# B&R Automation Studio project 305841_E00002_0 (part 2)

#### PBActions.st
```iecst
// For each button, check the state in the action.
// Call the action regardlesss of sate and check the state
// within the action rather than before calling in case there
// is something to do when the state is off.

// Ready. PB function not assigned
ACTION ProcessPb1 :
  IF owsPendant.PBStates[1] THEN
    // PB state is on ... process away
    ; // nothing to do
  ELSE
    // PB state is off ...
    ; // placeholder for future use
  END_IF;
END_ACTION

// Not assigned
ACTION ProcessPb2 :
  IF owsPendant.PBStates[2] THEN
    // PB state is on ... process away
    ; // nothing to do
  ELSE
    // PB state is off ...
    ; // placeholder for future use
  END_IF;
END_ACTION

// Set Zero
ACTION ProcessPb3 :
  IF owsPendant.PBStates[3] THEN
    // PB state is on ... depending on the axis, home the axis to zero.
    // The PB is a OS, so snapshot the axis selection and the home req.
    // Homing may take several scans, once kicked off, ignore selection
    // changes, PB changes, etc.
    axisSelection := owsPendant.AxisSelection;
    setZeroReq := TRUE;
  ELSE
    // PB state is off ...
    ; // placeholder for future use
  END_IF;
END_ACTION

// Axis Enable
ACTION ProcessPb4 :
  IF owsPendant.PBStates[4] THEN
    // PB state is on ... Send enable if drive is ready to be powered.
    // PB is OneShotted, and request only needs to be set, and is then cleared elsewhere
    axes[owsPendant.AxisSelection].Commands.EnableReq := axes[owsPendant.AxisSelection].Status.IsReadyToPowerOn;
  ELSE
    // PB state is off ...
    ; // placeholder for future use
  END_IF;
END_ACTION

// Axis Disable
ACTION ProcessPb5 :
  IF owsPendant.PBStates[5] THEN
    // PB state is on ... send disable if drive is powered on.
    // PB is OneShotted, and request only needs to be set, and is then cleared elsewhere
    axes[owsPendant.AxisSelection].Commands.DisableReq := axes[owsPendant.AxisSelection].Status.IsPoweredOn;
  ELSE
    // PB state is off ...
    ; // placeholder for future use
  END_IF;
END_ACTION

// Brake Off
ACTION ProcessPb6 :
  IF owsPendant.PBStates[6] THEN
    // PB state is on ... turn on brake release if the drive is disabled
    axes[owsPendant.AxisSelection].Commands.ReleaseBrakeReq := NOT axes[owsPendant.AxisSelection].Status.IsPoweredOn;
  ELSE
    // PB state is off ... turn off brake release
    axes[owsPendant.AxisSelection].Commands.ClearReleaseBrakeReq := TRUE;
    axes[owsPendant.AxisSelection].Commands.ReleaseBrakeReq := FALSE;
  END_IF;
END_ACTION

// Z Set SOC -- Axiz Z needs to be selected
ACTION ProcessPb7 :
  IF owsPendant.PBStates[7] AND owsPendant.AxisSelection = AD_Z THEN
    // PB state is on ... Set the current position to the Start Of Cut (SOC) position as long as the axis is homed.
    IF axes[AD_Z].Status.IsHomed THEN
      gr_CfgCurrent.zAxis.startOfCutPos := axes[AD_Z].Status.Position;
    END_IF;
  ELSE
    // PB state is off ...
    ; // placeholder for future use
  END_IF;
END_ACTION

// Z Set Load/Unload -- Axiz Z needs to be selected
ACTION ProcessPb8 :
  IF owsPendant.PBStates[8] AND owsPendant.AxisSelection = AD_Z THEN
    // PB state is on ... Set the current position to the load/unload position as long as the axis is homed.
    IF axes[AD_Z].Status.IsHomed THEN
      gr_CfgCurrent.zAxis.loadUnloadPos := axes[AD_Z].Status.Position;
    END_IF;
  ELSE
    // PB state is off ...
    ; // placeholder for future use
  END_IF;
END_ACTION

// Not assigned
ACTION ProcessPb9 :
  IF owsPendant.PBStates[9] THEN
    // PB state is on ... process away
    ;
  ELSE
    // PB state is off ...
    ; // placeholder for future use
  END_IF;
END_ACTION

ACTION SetZeroSeq :
  // The set zero sequence is started by PB3.
  // Handle the details here, just to the PB action is kept simple.
  // PB3 sets local axis selection and home req so changes during
  // homing are ignored.

  // Handle the req, and associated OS.
  // The OS is just so we can init values, and not keep resetting them
  // during homing

  IF NOT setZeroReq THEN
    // No Req, clear the OS
    homeSeqOS := FALSE;
  ELSIF setZeroReq AND NOT homeSeqOS THEN
    // Req and no OS, first time thru ...

    // Set the OS
    homeSeqOS := TRUE;

    // Now do the first time setup stuff ...

    // Now set the set zero offset based on the selected axis ... allow for different
    // algorithms based on axis
    IF axisSelection = AD_X THEN
      // TODO: Not sure how to handle X
      axes[axisSelection].MoveParameters.HomeParams.Position := 0.0;
    ELSIF axisSelection = AD_Y THEN
      // TODO: Not sure how to handle Y
      axes[axisSelection].MoveParameters.HomeParams.Position := 0.0;
    ELSIF axisSelection = AD_Z THEN
      // After homing, the desired position is zero + a possible offset
      axes[axisSelection].MoveParameters.HomeParams.Position :=  0.0;
    ELSIF axisSelection = AD_OUTER_ECCENTRIC THEN
      // Outer eccentric just gets homed to 0, no matter where it is, so there is no offset.
      axes[axisSelection].MoveParameters.HomeParams.Position := 0.0;
    ELSIF axisSelection = AD_INNER_ECCENTRIC THEN
      // After homing, the desired position is zero + a possible offset
      axes[axisSelection].MoveParameters.HomeParams.Position :=0.0;
    ELSIF axisSelection = AD_SPINDLE THEN
      // Spindle position isn't critical, so just home to zero
      axes[axisSelection].MoveParameters.HomeParams.Position := 0.0;
    END_IF;

    // Now set the home request for the selected axis
    axes[axisSelection].MoveParameters.HomeParams.Mode := mcHOMING_ABSOLUTE;
    axes[axisSelection].Commands.HomeReq := TRUE;

  ELSIF setZeroReq AND homeSeqOS THEN
    // Req and OS, doing while req is high
    // If the home command and req are both low, the homing is complete, successful or not.
    // If homing is successful, then set the 'isCalibrated' bits.
    IF NOT axes[axisSelection].Commands.HomeReq AND NOT axes[axisSelection].Commands.HomeCmd THEN
      IF axes[axisSelection].Status.IsHomed AND axes[axisSelection].Status.Position = 0.0 THEN
        // Home done and sucessful
        // Set the calibration bits based on selected axis
        IF axisSelection = AD_Z THEN
          gr_PartCurrent.isZCalibrated := TRUE;
        ELSIF axisSelection = AD_OUTER_ECCENTRIC THEN
          gr_PartCurrent.isOutECalibrated := TRUE;
        ELSIF axisSelection = AD_INNER_ECCENTRIC THEN
          gr_PartCurrent.isInECalibrated := TRUE;
        END_IF;
      END_IF;

      // All done, clear the req whether or not it was successful
      setZeroReq := FALSE;
    END_IF;
  END_IF;
END_ACTION

(*
ACTION SetZeroSeqOld :
  // The set zero sequence is started by PB3.
  // Handle the details here, just to the PB action is kept simple.
  // PB3 sets local axis selection and home req so changes during
  // homing are ignored.

  // Handle the req, and associated OS.
  // The OS is just so we can init values, and not keep resetting them
  // during homing

  // The actual homing is handled by the GaMot library function called outside this action.

  IF NOT setZeroReq THEN
    // No Req, clear the OS
    homeSeqOS := FALSE;
  ELSIF setZeroReq AND NOT homeSeqOS THEN
    // Req and no OS, first time thru ...

    // Set the OS
    homeSeqOS := TRUE;

    // Now do the first time setup stuff ...

    // Set the axis to the selected axis
    HomeAxisFb._I_Axis := ADR(axes[axisSelection]);

    // Now set the set zero offset based on the selected axis ... allow for different
    // algorithms based on axis
    IF axisSelection = AD_X THEN
      // TODO: Not sure how to handle X
      HomeAxisFb._I_Position := 0.0;
    ELSIF axisSelection = AD_Y THEN
      // TODO: Not sure how to handle Y
      HomeAxisFb._I_Position := 0.0;
    ELSIF axisSelection = AD_Z THEN
      // After homing, the desired position is zero + a possible offset
      HomeAxisFb._I_Position :=  gr_CfgCurrent.zAxis.setZeroOffset;;
    ELSIF axisSelection = AD_OUTER_ECCENTRIC THEN
      // Outer eccentric just gets homed to 0, no matter where it is, so there is no offset.
      HomeAxisFb._I_Position := 0.0;
    ELSIF axisSelection = AD_INNER_ECCENTRIC THEN
      // After homing, the desired position is zero + a possible offset
      HomeAxisFb._I_Position := gr_CfgCurrent.cuttingHead.setZeroOffset;
    ELSIF axisSelection = AD_SPINDLE THEN
      // Spindle position isn't critical, so just home to zero
      HomeAxisFb._I_Position := 0.0;
    END_IF;

  ELSIF setZeroReq AND homeSeqOS THEN
    // Req and OS, doing while req is high
    // The fb is always called below, and the enable is based on the setZeroReq.
    // Monitor the output of the FB here. It should end sucessfully or in error
    IF fbHomeAbs._O_Done AND NOT fbHomeAbs._O_Error THEN
      // Homing done, and no error -- Success!!
      // Clear the home req and consider the axis homed.
      setZeroReq := FALSE;
      // Set the calibration bits based on selected axis
      IF axisSelection = AD_Z THEN
        gr_PartCurrent.isZCalibrated := TRUE;
      ELSIF axisSelection = AD_OUTER_ECCENTRIC THEN
        gr_PartCurrent.isOutECalibrated := TRUE;
      ELSIF axisSelection = AD_INNER_ECCENTRIC THEN
        gr_PartCurrent.isInECalibrated := TRUE;
      END_IF;
    ELSIF fbHomeAbs._O_Done AND fbHomeAbs._O_Error THEN
      // Homing done, but in error :(
      // Clear the home req
      setZeroReq := FALSE;
      // Clear the calibration bits based on selected axis
      IF axisSelection = AD_Z THEN
        gr_PartCurrent.isZCalibrated := FALSE;
      ELSIF axisSelection = AD_OUTER_ECCENTRIC THEN
        gr_PartCurrent.isOutECalibrated := FALSE;
      ELSIF axisSelection = AD_INNER_ECCENTRIC THEN
        gr_PartCurrent.isInECalibrated := FALSE;
      END_IF;
    ELSE
      // fb not done ... fb must be busy ... nothing to do.
      // Keep for future expansion
      ;
    END_IF;

  END_IF;

END_ACTION

ACTION HomeInPosSeqOld :
  // The home sequence is started by PB3.
  // Handle the details here, just to the PB action is kept simple.
  // PB3 sets local axis selection and home req so changes during
  // homing are ignored.

  // Handle the req, and associated OS.
  // The OS is just so we can init values, and not keep resetting them
  // during homing

  // The actual homing is handled by the GaMot library function called outside this action.

  IF NOT homeInPosReq THEN
    // No Req, clear the OS
    homeSeqOS := FALSE;
  ELSIF homeInPosReq AND NOT homeSeqOS THEN
    // Req and no OS, first time thru ...

    // Set the OS
    homeSeqOS := TRUE;

    // Now do the first time setup stuff ...

    // Set the axis to the selected axis
    fbHomeAbs._I_Axis := ADR(axes[axisSelection]);

    // Now set the desired poition to the axis position
    fbHomeAbs._I_Position := axes[axisSelection].Status.Position;

  ELSIF homeInPosReq AND homeSeqOS THEN
    // Req and OS, doing while req is high
    // The fb is always called below, and the enable is based on the homeInPosReq.
    // Monitor the output of the FB here. It should end sucessfully or in error
    IF fbHomeAbs._O_Done AND NOT fbHomeAbs._O_Error THEN
      // Homing done, and no error -- Success!!
      // Clear the home req and consider the axis homed.
      homeInPosReq := FALSE;

      // Other success stuff here ...

    ELSIF fbHomeAbs._O_Done AND fbHomeAbs._O_Error THEN
      // Homing done, but in error :(
      // Clear the home req
      homeInPosReq := FALSE;

      // Other error stuff here ...

    ELSE
      // fb not done ... fb must be busy ... nothing to do.
      // Keep for future expansion
      ;
    END_IF;

  END_IF;

 END_ACTION
*)
```

### Program Logical/PlcLogic/CuttingFluidVFD (IEC)

#### Variables.var
```iecst
VAR

  almMask : UDINT;
  tmrCfFlowOk : TON; (* flow established timer *)
  timeCfFlowOk : TIME;

END_VAR
```

#### Action.st
```iecst
ACTION ProcessAlarms :
  // Alarm Enable/disable. These are permanent, but include here to easily make them dynamic.
  // Tank level
  gr_AI_LT_CFTankLevel_Params.AlmEnable := FALSE; // not fitted.
  // Flow
  gr_AI_FT_CFFlow_Params.AlmEnable := FALSE; // not fitted
  // Level switch
  gr_DI_LSL_CFTank_Params.AlmEnable := FALSE; // not fitted
  // Locator
  gr_DI_ZS_CFTankLocator_Params.AlmEnable:= TRUE;

  // Pressure and flow sensors -- enable while pump is running
  gr_AI_PT_CFPumpOutlet_Params.AlmEnable := cfVfd.isRunning;
  gr_AI_PT_CFFilterOutlet_Params.AlmEnable := cfVfd.isRunning;
  gr_AI_DP_CFFilter_Params.AlmEnable := cfVfd.isRunning;
  gr_AI_FT_CFFlow_Params.AlmEnable := cfVfd.isRunning;

  // Put alarm status into structure
  // isLocated
  cfVfd.isLocated := DI_ZS_CFTankLocator.alms = GAPIO_ALARM_NONE;

  // Level switch
  cfVfd.isAlmLoLvlSw := DI_LSL_CFTank.alms <> GAPIO_ALARM_NONE;

  // Flow
  // consider alarm on range, channel or lo lo alms
  almMask := 	GAPIO_ALARM_RANGEHI OR GAPIO_ALARM_RANGELO OR GAPIO_ALARM_CHANNEL OR GAPIO_ALARM_LOLO;
  cfVfd.isAlmLoFlow := (AI_FT_CFFlow.alms AND almMask) <> 0;
  // consider warning on lo alm
  almMask := GAPIO_ALARM_LO;
  cfVfd.isWarnLoFlow := (AI_FT_CFFlow.alms AND almMask) <> 0;

  // Fluid Level
  // consider alarm on range, channel or lo lo alms
  almMask := 	GAPIO_ALARM_RANGEHI OR GAPIO_ALARM_RANGELO OR GAPIO_ALARM_CHANNEL OR GAPIO_ALARM_LOLO;
  cfVfd.isAlmLoFluid := (AI_LT_CFTankLevel.alms AND almMask) <> 0;
  // consider warning on lo alm
  almMask := 	GAPIO_ALARM_LO;
  cfVfd.isWarnLoFluid := (AI_LT_CFTankLevel.alms AND almMask) <> 0;

  // Pump Outlet pressure
  // consider alarm on hi range, channel or hi hi alms
  almMask := 	GAPIO_ALARM_RANGEHI OR GAPIO_ALARM_CHANNEL OR GAPIO_ALARM_HIHI;
  cfVfd.isAlmHiOutletPressure := (AI_PT_CFPumpOutlet.alms AND almMask) <> 0;
  // consider alarm on range, channel or lo lo alms
  almMask := 	GAPIO_ALARM_RANGELO OR GAPIO_ALARM_LOLO;
  cfVfd.isAlmLoOutletPressure := (AI_PT_CFPumpOutlet.alms AND almMask) <> 0;
  // consider warning on lo alm
  almMask := 	GAPIO_ALARM_LO;
  cfVfd.isWarnLoOutletPressure := (AI_PT_CFPumpOutlet.alms AND almMask) <> 0;
  // consider warning on hi alm
  almMask := 	GAPIO_ALARM_HI;
  cfVfd.isWarnHiOutletPressure := (AI_PT_CFPumpOutlet.alms AND almMask) <> 0;

  // Hi Filter DP -- channel and range will trigger hi and low
  almMask := 	GAPIO_ALARM_RANGEHI OR GAPIO_ALARM_RANGELO OR GAPIO_ALARM_CHANNEL OR GAPIO_ALARM_HI;
  cfVfd.isWarnHiFilterDp := (AI_DP_CFFilter.alms AND almMask) <> 0;
  // Lo Filter DP -- channel and range will trigger hi and low
  almMask := 	GAPIO_ALARM_RANGEHI OR GAPIO_ALARM_RANGELO OR GAPIO_ALARM_CHANNEL OR GAPIO_ALARM_LO;
  cfVfd.isWarnLoFilterDp := (AI_DP_CFFilter.alms AND almMask) <> 0;

  // Alarm and warning summaries
  cfVfd.isWarnSummary := cfVfd.isWarnLoFlow OR cfVfd.isWarnLoFluid OR
  cfVfd.isWarnLoOutletPressure OR cfVfd.isWarnHiOutletPressure OR
  cfVfd.isWarnLoFilterDp OR cfVfd.isWarnHiFilterDp;

  cfVfd.isAlmSummary := cfVfd.isAlmLoFlow OR cfVfd.isAlmLoLvlSw OR
  cfVfd.isAlmLoFluid OR cfVfd.isAlmLoOutletPressure OR cfVfd.isAlmHiOutletPressure;

END_ACTION
```

#### Main.st
```iecst
PROGRAM _INIT

  // Flow established time
  timeCfFlowOk := T#5s;

END_PROGRAM

PROGRAM _CYCLIC

  // Process the alarms
  ProcessAlarms;

  cfVfd.isAllowedToStart :=
    (operatingMode.OperatingMode = OM_MANUAL_MODE OR
    operatingMode.OperatingMode = OM_PENDANT_MODE OR
    operatingMode.OperatingMode = OM_PRODUCTION_MODE) AND
    axes[AD_CF_VFD].Status.IsPoweredOn AND
    axes[AD_CF_VFD].Status.IsHomed AND
    cfVfd.isLocated AND
    NOT cfVfd.isAlmLoLvlSw AND NOT cfVfd.isAlmLoFluid;

  cfVfd.isAllowedToRun :=
    (operatingMode.OperatingMode = OM_MANUAL_MODE OR
    operatingMode.OperatingMode = OM_PENDANT_MODE OR
    operatingMode.OperatingMode = OM_PRODUCTION_MODE) AND
    axes[AD_CF_VFD].Status.IsPoweredOn AND
    axes[AD_CF_VFD].Status.IsHomed AND
    cfVfd.isLocated AND
    NOT cfVfd.isAlmLoLvlSw AND NOT cfVfd.isAlmLoFluid AND
    NOT cfVfd.isAlmLoFlow AND NOT cfVfd.isAlmLoOutletPressure AND
    NOT cfVfd.isAlmHiOutletPressure;

  // Map the axis status to the cf structure to get a running bit
  cfVfd.isRunning := axes[AD_CF_VFD].Status.IsMoveActive;

  // Determine when good flow is established -- time delay no flow problems
  tmrCfFlowOk(IN:= cfVfd.isRunning AND NOT cfVfd.isAlmLoFlow, PT:= timeCfFlowOk);
  cfVfd.isFlowEstablished := tmrCfFlowOk.Q;

END_PROGRAM

PROGRAM _EXIT
	(* Insert code here *)

END_PROGRAM
```

### Program Logical/PlcLogic/OmSafeDev (IEC) - Operating Mode State Machine

#### OmSafeDev.typ - Local data types
```iecst
TYPE
  (* Machine specific HMI axis requests. Intended to have one of these structures per axis. *)
  sHmiAxisReqs : STRUCT
    (* Boolean requests in this section. *)
    (* (none *)
    (* numerical requests *)
    (* (none *)
    (* hmi move type and direction selection related *)
    absMoveEnable : BOOL := TRUE; (* allow move type selection by default *)
    relMoveEnable : BOOL := TRUE;
    velMoveEnable : BOOL := TRUE;
    directionPosEnable : BOOL := TRUE; (* allow direction selection by default *)
    directionNegEnable : BOOL := TRUE;
    directionShortestEnable : BOOL := TRUE;
    moveDistanceEnable : BOOL := TRUE; (* enable params by default *)
    movePositionEnable : BOOL := TRUE;
    shiftEnable : BOOL := FALSE; (* coordinated axis shift enabled *)
    moveDesignation: DINT := -1; (* -1 is no selection *)
    direction: DINT := -1; (* -1 is no selection *)
    (* axis designation. Two different data types for convenience. *)
    axisNo : USINT := 0; (* default to initial so setting a value can be detected. USINT for easy use in loops *)
    axisDesignation : eAXIS_DESIGNATION := AD_UNKNOWN; (* default to initial so setting a value can be detected *)
  END_STRUCT;

  (* Machine specific HMI process requests. Intended to have one of these per machine or otherwise as needed, but not per axis. *)
  sHmiProcessReqs : STRUCT
    (* Boolean requests in this section. *)
    (* NOTE/CAUTION These request bits may get cleared/copied by memcpy/memclr
    So be careful about adding boolean requests outside of this section.
    See ClearManualReqs action for example, in OmSaveDev program.
    Bool requests above zReqMoveUpLimit won't get auto cleared *)
    zReqMoveUpLimit : BOOL := FALSE;
    zReqMoveDownLimit : BOOL := FALSE;
    zReqMoveLoadUnload : BOOL := FALSE;
    zReqMoveSoc : BOOL := FALSE;
    cuttingHeadMoveReqRetract : BOOL := FALSE;
    (* NOTE/CAUTION Bool requests below cuttingHeadMoveReqRetract won't get auto cleared *)
    (* numerical requests *)
    cuttingHeadReqDepth : LREAL := 0.0;
  END_STRUCT;

END_TYPE
```

#### OmSafeDev.var - Local variables
```iecst
VAR CONSTANT

END_VAR

VAR

  (* info from safety controller *)
  fs_AllSMsOk : BOOL;
  fs_EmoCmd : BOOL; (* H:Ok, L:EMO *)
  fs_EmoOwsActive : BOOL; (* H:Ok, L: EMO *)
  fs_EmoOwsOk : BOOL; (* H:Wiring Ok, L:Error *)
  fs_InSafeMode : BOOL; (* H:InSafeMode, L: Not in safe mode *)
  fs_KeyswitchInRun : BOOL; (* H:Run Pos, L: Not in run pos *)
  fs_KeyswitchOk : BOOL; (* H:Wiring Ok, L:Error *)
  fs_StartPbActive : BOOL; (* H:Start Req, L: Not pressed *)
  fs_StartPbOk : BOOL; (* H:Wiring Ok, L:Error *)
  fs_StopPbActive : BOOL; (* H: Allow Run, L: Stop *)
  fs_StopPbOk : BOOL; (* H:Wiring Ok, L:Error *)
  fs_CfGateClosed : BOOL; (* H:Closed, L: Open *)
  fs_CfGateClosedLocked : BOOL; (* H:Closed and locked(Ok), L: Open and/or unlocked *)
  fs_CfGateClosedOk : BOOL; (* H:Wiring Ok, L: Error *)

  (* info to safety controller *)
  ts_ResetEStop : BOOL;
  ts_ResetSafeMC : BOOL;
  ts_InEmoMode : BOOL;
  ts_InSafeMode : BOOL;
  ts_InPendantMode : BOOL;

  (* cycle start/stop req *)
  tmrReqStartPulse : TP;
  tmrReqStopPulse : TP;

  (* EMO Reset *)
  timeEStopResetAllow : TIME;
  eStopResetAllowSecRemain : DINT;
  tmrEStopResetAllow : TON;
  timeResetPulse : TIME;
  tmrResetPulse : TP;

  (* HMI process specific, machine specific, and axis requests *)
  hmiProcessReqs : sHmiProcessReqs; (* process specific reqs *)
  hmiMachineAxisReqs : ARRAY[0..AXIS_COUNT] OF sHmiAxisReqs; (* machine specific requests that get turned into library reqs *)
  hmiLibraryAxisReqs : ARRAY[0..AXIS_COUNT] OF sMot_HmiAxisReqs; (* standard/basic requests handled by the library *)

  (* pointers used for memcpy/memset *)
  pSrc :  UDINT;
  pDest :  UDINT;
  byteCount :  UDINT;
  nxtAddr :  UDINT;

  (* axis index *)
  axisNo : DINT;

  (* fb to process Reqs *)
  procHmiProcessReqs : fbHandleHmiProcessReqs;
  procManualAxisReqsSpindle : fbHandleHmiAxisReq;
  procManualAxisReqsOutE : fbHandleHmiAxisReq;
  procManualAxisReqsInE : fbHandleHmiAxisReq;
  procManualAxisReqsZ : fbHandleHmiAxisReq;
  procManualAxisReqsHw : fbHandleHmiAxisReq;
  procManualAxisReqsCfVfd : fbHandleHmiAxisReq;
END_VAR
```

#### Init.st
```iecst
PROGRAM _INIT

  // TODO: Security levels. For now just set as operator so OM SM can be programmed
  operatingMode.SecurityLevel := SL_OPERATOR;

  // EMO Reset time
  timeEStopResetAllow := T#10s;
  timeResetPulse := T#1s;

  // Init to create variables
  // If values are only mapped, and not used in logic anywhere, the compiler does not
  // create them. They are not available to
  // the HMI, and the compiler also complains about
  // them being declared but not used
  fs_AllSMsOk := FALSE;
  fs_EmoCmd := FALSE;
  fs_EmoOwsActive := FALSE;
  fs_EmoOwsOk := FALSE;
  // pendant signals are mapped into pendant structure
  // fs_EmoPendantActive := FALSE;
  // fs_EmoPendantOk := FALSE;
  // fs_AllowPendantMoves := FALSE;
  fs_KeyswitchInRun := FALSE;
  fs_KeyswitchOk := FALSE;
  fs_InSafeMode := FALSE;
  fs_StartPbActive := FALSE;
  fs_StartPbOk := FALSE;
  fs_StopPbActive := FALSE;
  fs_StopPbOk := FALSE;
  fs_CfGateClosedLocked := FALSE;
  fs_CfGateClosedOk := FALSE;

  ts_ResetEStop := FALSE;
  ts_ResetSafeMC := FALSE;

  // Init process req fb
  procHmiProcessReqs._I_ProcessReqs := ADR(hmiProcessReqs);
  procHmiProcessReqs._I_pLibraryAxesReqs:= ADR(hmiLibraryAxisReqs); // Start of array of sMot_HmiAxisReqs

  // Init manual mode requests
  hmiLibraryAxisReqs[AD_SPINDLE].axisNo := DINT_TO_USINT(AD_SPINDLE);
  hmiMachineAxisReqs[AD_SPINDLE].axisNo := DINT_TO_USINT(AD_SPINDLE);
  hmiMachineAxisReqs[AD_SPINDLE].axisDesignation := AD_SPINDLE;
  procManualAxisReqsSpindle._I_Axis := ADR(axes[AD_SPINDLE]);
  procManualAxisReqsSpindle._I_SlaveAxis := ADR(axes[axes[AD_SPINDLE].CouplingParameters.SlaveAxisNo]);
  procManualAxisReqsSpindle._I_LibraryAxisReqs := ADR(hmiLibraryAxisReqs[AD_SPINDLE]);
  procManualAxisReqsSpindle._I_MachineAxisReqs := ADR(hmiMachineAxisReqs[AD_SPINDLE]);
  procManualAxisReqsSpindle._I_AxisPositionLimits := ADR(gr_AxisPositionLimits[AD_SPINDLE]);

  // Outer Eccentric
  hmiLibraryAxisReqs[AD_OUTER_ECCENTRIC].axisNo := DINT_TO_USINT(AD_OUTER_ECCENTRIC);
  hmiMachineAxisReqs[AD_OUTER_ECCENTRIC].axisNo := DINT_TO_USINT(AD_OUTER_ECCENTRIC);
  hmiMachineAxisReqs[AD_OUTER_ECCENTRIC].axisDesignation := AD_OUTER_ECCENTRIC;
  procManualAxisReqsOutE._I_Axis := ADR(axes[AD_OUTER_ECCENTRIC]);
  procManualAxisReqsOutE._I_SlaveAxis := ADR(axes[axes[AD_OUTER_ECCENTRIC].CouplingParameters.SlaveAxisNo]);
  procManualAxisReqsOutE._I_LibraryAxisReqs := ADR(hmiLibraryAxisReqs[AD_OUTER_ECCENTRIC]);
  procManualAxisReqsOutE._I_MachineAxisReqs:= ADR(hmiMachineAxisReqs[AD_OUTER_ECCENTRIC]);
  procManualAxisReqsOutE._I_AxisPositionLimits := ADR(gr_AxisPositionLimits[AD_OUTER_ECCENTRIC]);

  // Inner Eccentric
  hmiLibraryAxisReqs[AD_INNER_ECCENTRIC].axisNo := DINT_TO_USINT(AD_INNER_ECCENTRIC);
  hmiMachineAxisReqs[AD_INNER_ECCENTRIC].axisNo := DINT_TO_USINT(AD_INNER_ECCENTRIC);
  hmiMachineAxisReqs[AD_INNER_ECCENTRIC].axisDesignation := AD_INNER_ECCENTRIC;
  procManualAxisReqsInE._I_Axis := ADR(axes[AD_INNER_ECCENTRIC]);
  procManualAxisReqsInE._I_SlaveAxis := ADR(axes[axes[AD_INNER_ECCENTRIC].CouplingParameters.SlaveAxisNo]);
  procManualAxisReqsInE._I_LibraryAxisReqs := ADR(hmiLibraryAxisReqs[AD_INNER_ECCENTRIC]);
  procManualAxisReqsInE._I_MachineAxisReqs := ADR(hmiMachineAxisReqs[AD_INNER_ECCENTRIC]);
  procManualAxisReqsInE._I_AxisPositionLimits := ADR(gr_AxisPositionLimits[AD_INNER_ECCENTRIC]);

  // Z
  hmiLibraryAxisReqs[AD_Z].axisNo := DINT_TO_USINT(AD_Z);
  hmiMachineAxisReqs[AD_Z].axisNo := DINT_TO_USINT(AD_Z);
  hmiMachineAxisReqs[AD_Z].axisDesignation := AD_Z;
  procManualAxisReqsZ._I_Axis := ADR(axes[AD_Z]);
  procManualAxisReqsZ._I_SlaveAxis := ADR(axes[axes[AD_Z].CouplingParameters.SlaveAxisNo]);
  procManualAxisReqsZ._I_LibraryAxisReqs := ADR(hmiLibraryAxisReqs[AD_Z]);
  procManualAxisReqsZ._I_MachineAxisReqs := ADR(hmiMachineAxisReqs[AD_Z]);
  procManualAxisReqsZ._I_AxisPositionLimits := ADR(gr_AxisPositionLimits[AD_Z]);

  // Handwheel (Axis 7)
  hmiLibraryAxisReqs[AD_HANDWHEEL].axisNo := DINT_TO_USINT(AD_HANDWHEEL);
  hmiMachineAxisReqs[AD_HANDWHEEL].axisNo := DINT_TO_USINT(AD_HANDWHEEL);
  hmiMachineAxisReqs[AD_HANDWHEEL].axisDesignation := AD_HANDWHEEL;
  procManualAxisReqsHw._I_Axis := ADR(axes[AD_HANDWHEEL]);
  procManualAxisReqsHw._I_SlaveAxis := ADR(axes[axes[AD_HANDWHEEL].CouplingParameters.SlaveAxisNo]);
  procManualAxisReqsHw._I_LibraryAxisReqs := ADR(hmiLibraryAxisReqs[AD_HANDWHEEL]);
  procManualAxisReqsHw._I_MachineAxisReqs := ADR(hmiMachineAxisReqs[AD_HANDWHEEL]);
  procManualAxisReqsHw._I_AxisPositionLimits := ADR(gr_AxisPositionLimits[AD_HANDWHEEL]);

  // Cutting fluid VFD (Axis 8)
  hmiLibraryAxisReqs[AD_CF_VFD].axisNo := DINT_TO_USINT(AD_CF_VFD);
  hmiMachineAxisReqs[AD_CF_VFD].axisNo := DINT_TO_USINT(AD_CF_VFD);
  hmiMachineAxisReqs[AD_CF_VFD].axisDesignation := AD_CF_VFD;
  procManualAxisReqsCfVfd._I_Axis := ADR(axes[AD_CF_VFD]);
  procManualAxisReqsCfVfd._I_SlaveAxis := ADR(axes[axes[AD_CF_VFD].CouplingParameters.SlaveAxisNo]);
  procManualAxisReqsCfVfd._I_LibraryAxisReqs := ADR(hmiLibraryAxisReqs[AD_CF_VFD]);
  procManualAxisReqsCfVfd._I_MachineAxisReqs := ADR(hmiMachineAxisReqs[AD_CF_VFD]);
  procManualAxisReqsCfVfd._I_AxisPositionLimits := ADR(gr_AxisPositionLimits[AD_CF_VFD]);

  // Clear reqs that may result in motion or physical changes to an axis
  ClearMotionReqs;
  // Clear other requests
  ClearNonMotionReqs;

END_PROGRAM
```

#### OmSafeDev.sfc - Cyclic code
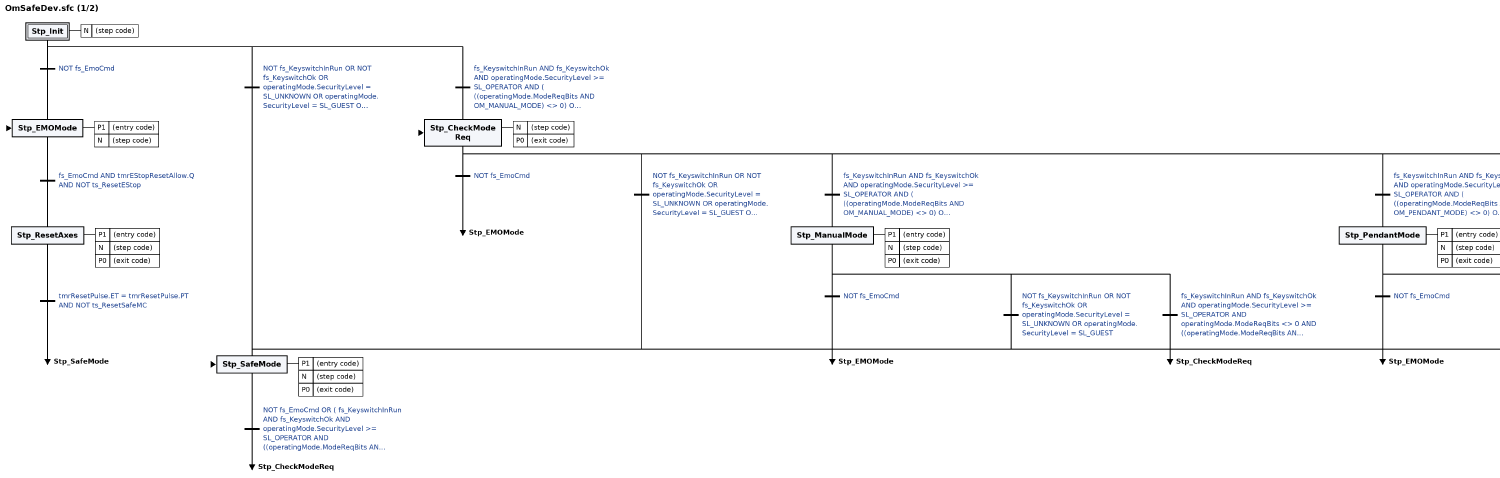
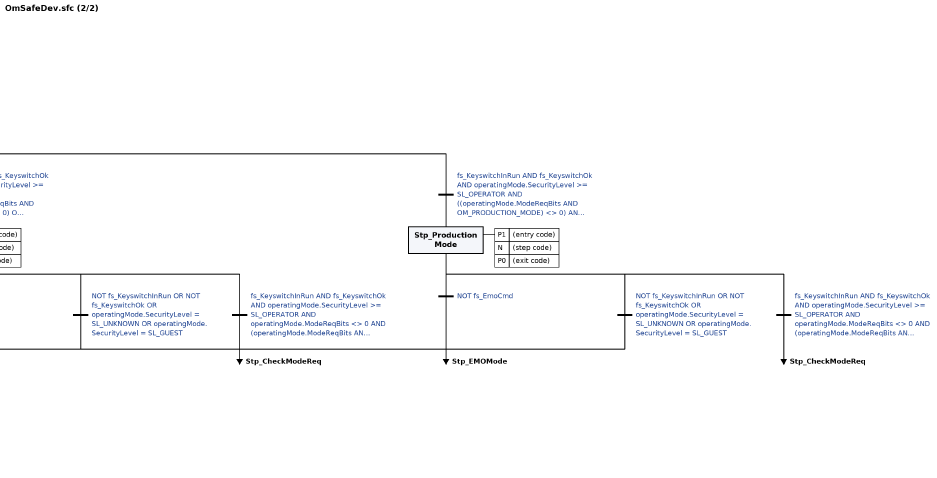
```iecst
PROGRAM _CYCLIC
INITIAL_STEP Stp_Init:
// Set Operating State
operatingMode.OperatingMode := OM_INITIAL;

END_STEP
TRANSITION EMO Cmd FROM Stp_Init TO Stp_EMOMode:=
// EStop command from safety plc H:Ok, L:EMO
NOT fs_EmoCmd
END_TRANSITION
TRANSITION keyswich in safe, not ok or bad SL or no mode req FROM Stp_Init TO Stp_SafeMode:=
// Keyswitch not in run or not okay
NOT fs_KeyswitchInRun OR
NOT fs_KeyswitchOk OR
// or not adequate security level
operatingMode.SecurityLevel = SL_UNKNOWN OR
operatingMode.SecurityLevel = SL_GUEST OR
// Or a mode isnt' being requested.
// Go to safe initially if all else is okay so a mode must be chosen
operatingMode.ModeReqBits = 0
END_TRANSITION
TRANSITION keyswitch in run and SL FROM Stp_Init TO Stp_CheckModeReq:=
// Keyswitch in run and adequate security level
fs_KeyswitchInRun AND
fs_KeyswitchOk AND
operatingMode.SecurityLevel >= SL_OPERATOR AND
// and a mode is requested
(
((operatingMode.ModeReqBits AND OM_MANUAL_MODE) <> 0) OR
((operatingMode.ModeReqBits AND OM_PENDANT_MODE) <> 0) OR
((operatingMode.ModeReqBits AND OM_PRODUCTION_MODE) <> 0)
)

END_TRANSITION
STEP Stp_CheckModeReq:
// This is a transition state. The state machine should not stay here, so don't
// set the mode upon entry. The mode in fact cannot be changed, as the current value is
// is used to transition back into the same state if a request was made but not granted
// for example production mode req but gate isn't shut.

// Clear reqs that may result in motion or physical changes to an axis
ClearMotionReqs;
// Clear other requests
ClearNonMotionReqs;

// Axis permit and other permissives
OtherModeAxisPermits;
ModeIndependentPermissions;
END_STEP
EXIT_ACTION
// Clear the request bits when leaving
operatingMode.ModeReqBits := 0;
END_ACTION
TRANSITION EMO Cmd FROM Stp_CheckModeReq TO Stp_EMOMode:=
// EStop command from safety plc H:Ok, L:EMO
NOT fs_EmoCmd
END_TRANSITION
(* @SFCISJUMP := 'Stp_EMOMode' *)
TRANSITION key not in run or bad SL or prod mode but not allowed FROM Stp_CheckModeReq TO Stp_SafeMode:=
// Keyswitch not in run or not okay, or not adequate security level
NOT fs_KeyswitchInRun OR
NOT fs_KeyswitchOk OR
operatingMode.SecurityLevel = SL_UNKNOWN OR
operatingMode.SecurityLevel = SL_GUEST OR
// or requested production mode but the gate isn't closed, so stay here in safe mode
(((operatingMode.ModeReqBits AND OM_PRODUCTION_MODE) <> 0) AND NOT fs_CfGateClosed AND operatingMode.OperatingMode = OM_SAFE_MODE)

END_TRANSITION
TRANSITION req manual mode or prod mode but not allowed FROM Stp_CheckModeReq TO Stp_ManualMode:=
// Keyswitch in run and adequate security level
fs_KeyswitchInRun AND
fs_KeyswitchOk AND
operatingMode.SecurityLevel >= SL_OPERATOR AND
(
// Req Manual Mode
((operatingMode.ModeReqBits AND OM_MANUAL_MODE) <> 0) OR
// or requested production mode but the gate isn't closed, so stay here in manual mode
(((operatingMode.ModeReqBits AND OM_PRODUCTION_MODE) <> 0) AND NOT fs_CfGateClosed AND operatingMode.OperatingMode = OM_MANUAL_MODE)
)

END_TRANSITION
STEP Stp_ManualMode:
// Block mode request for current mode, but keep the others
// This prevents it from being seen as a request
operatingMode.ModeReqBits := operatingMode.ModeReqBits AND NOT OM_MANUAL_MODE; (* bit 4 clear *)

// Axis permit and other permissives
ManualModeAxisPermits;
ModeIndependentPermissions;

// Pulse the Reset SafeMC on request.
// This allows the reset of the safety enable instructions in the
// SafePLC while the system is not in EMO mode.
// The SafeMC reset sometimes isn't effective unless the axis is otherwise allowed to be powered.
tmrResetPulse(IN:= operatingMode.ReqEmoReset);
ts_ResetSafeMC := tmrResetPulse.Q;
operatingMode.ReqEmoReset := FALSE;

// Clear production start/stop cycle
operatingMode.ReqCycleStart := FALSE;
operatingMode.ReqCycleStop := FALSE;
operatingMode.HmiReqCycleStart := FALSE;
operatingMode.HmiReqCycleStop:= FALSE;

// Process manual requests
// Inputs set in init. This fb looks for a rising edge on the HMI move request, and
// one-shots the axis move requests. It is inteneded to be run on every scan,
// at least while in manual mode.
procManualAxisReqsSpindle();
procManualAxisReqsOutE();
procManualAxisReqsInE();
procManualAxisReqsZ();
procManualAxisReqsHw();
procManualAxisReqsCfVfd();
END_STEP
ENTRY_ACTION
// Set Operating State
operatingMode.OperatingMode := OM_MANUAL_MODE;
// To Safety PLC
ts_InManualMode := TRUE;

// Reset pulse timer
tmrResetPulse(IN:= FALSE, PT:= timeResetPulse);

// Clear reqs that may result in motion or physical changes to an axis
ClearMotionReqs;
// Clear other requests
ClearNonMotionReqs;

// Init fb with low reqs so rising edge detection is ready
procManualAxisReqsSpindle();
procManualAxisReqsOutE();
procManualAxisReqsInE();
procManualAxisReqsZ();
procManualAxisReqsHw();
procManualAxisReqsCfVfd();
END_ACTION
EXIT_ACTION
// To Safety PLC
ts_InManualMode := FALSE;

// Clear reqs that may result in motion or physical changes to an axis
ClearMotionReqs;
// Clear other requests
ClearNonMotionReqs;

// Init fb with low reqs so rising edge detection is ready
procManualAxisReqsSpindle();
procManualAxisReqsOutE();
procManualAxisReqsInE();
procManualAxisReqsZ();
procManualAxisReqsHw();
procManualAxisReqsCfVfd();
END_ACTION
TRANSITION EMO Cmd FROM Stp_ManualMode TO Stp_EMOMode:=
// EStop command from safety plc H:Ok, L:EMO
NOT fs_EmoCmd
END_TRANSITION
(* @SFCISJUMP := 'Stp_EMOMode' *)
TRANSITION key not in run or bad SL FROM Stp_ManualMode TO Stp_SafeMode:=
// Keyswitch not in run or not okay, or not adequate security level
NOT fs_KeyswitchInRun OR
NOT fs_KeyswitchOk OR
operatingMode.SecurityLevel = SL_UNKNOWN OR
operatingMode.SecurityLevel = SL_GUEST
END_TRANSITION
TRANSITION req mode change FROM Stp_ManualMode TO Stp_CheckModeReq:=
// Keyswitch in run and adequate security level
fs_KeyswitchInRun AND
fs_KeyswitchOk AND
operatingMode.SecurityLevel >= SL_OPERATOR AND
// Req mode change (req other than current mode)
operatingMode.ModeReqBits <> 0 AND
((operatingMode.ModeReqBits AND OM_MANUAL_MODE) = 0)

END_TRANSITION
(* @SFCISJUMP := 'Stp_CheckModeReq' *)
TRANSITION req pendant mode or prod mode but not allowed FROM Stp_CheckModeReq TO Stp_PendantMode:=
// Keyswitch in run and adequate security level
fs_KeyswitchInRun AND
fs_KeyswitchOk AND
operatingMode.SecurityLevel >= SL_OPERATOR AND
(
// Req Pendant Mode
((operatingMode.ModeReqBits AND OM_PENDANT_MODE) <> 0) OR
// or requested production mode but the gate isn't closed, so stay here in pendant mode
(((operatingMode.ModeReqBits AND OM_PRODUCTION_MODE) <> 0) AND NOT fs_CfGateClosed AND operatingMode.OperatingMode = OM_PENDANT_MODE)
)

END_TRANSITION
STEP Stp_PendantMode:
// Block mode request for current mode, but keep the others
// This prevents it from being seen as a request
operatingMode.ModeReqBits := operatingMode.ModeReqBits AND NOT OM_PENDANT_MODE; (* bit 5 clear *)

// Axis permit and other permissives
PendantModeAxisPermits;
ModeIndependentPermissions;

// Clear process reqs
ClearProcessReqs;

// Pulse the Reset SafeMC on request.
// This allows the reset of the safety enable instructions in the
// SafePLC while the system is not in EMO mode.
// The SafeMC reset sometimes isn't effective unless the axis is otherwise allowed to be powered.
tmrResetPulse(IN:= operatingMode.ReqEmoReset);
ts_ResetSafeMC := tmrResetPulse.Q;
operatingMode.ReqEmoReset := FALSE;

// Clear production start/stop cycle
operatingMode.ReqCycleStart := FALSE;
operatingMode.ReqCycleStop := FALSE;
operatingMode.HmiReqCycleStart := FALSE;
operatingMode.HmiReqCycleStop:= FALSE;

// Use the gear ratio coming from the pendant for the hmi request strucure.
// It is the hmi request structure values that will get sent to the axis.
hmiLibraryAxisReqs[AD_HANDWHEEL].gearRatioNumerator := owsPendant.GearRatioNumerator;
hmiLibraryAxisReqs[AD_HANDWHEEL].gearRatioDenominator := owsPendant.GearRatioDenominator;

// Process manual requests -- Allow these in pendant mode.
// Inputs set in init. This fb looks for a rising edge on the HMI move request, and
// one-shots the axis move requests. It is inteneded to be run on every scan,
// at least while in manual mode.
procManualAxisReqsSpindle();
procManualAxisReqsOutE();
procManualAxisReqsInE();
procManualAxisReqsZ();
procManualAxisReqsHw();
procManualAxisReqsCfVfd();

END_STEP
ENTRY_ACTION
// Set Operating State
operatingMode.OperatingMode := OM_PENDANT_MODE;
// To Safety PLC
ts_InPendantMode := TRUE;

// Reset pulse timer
tmrResetPulse(IN:= FALSE, PT:= timeResetPulse);

// Disable enabled axes on entry into pendant mode -- allows starting from the same point
FOR axisNo := 1 TO AXIS_COUNT DO
  axes[axisNo].Commands.DisableReq := axes[axisNo].Status.IsPoweredOn;
END_FOR;

// Clear reqs that may result in motion or physical changes to an axis
ClearMotionReqs;
// Clear other requests
ClearNonMotionReqs;

// Init fb with low reqs so rising edge detection is ready
procManualAxisReqsSpindle();
procManualAxisReqsOutE();
procManualAxisReqsInE();
procManualAxisReqsZ();
procManualAxisReqsHw();
procManualAxisReqsCfVfd();

END_ACTION
EXIT_ACTION
// To Safety PLC
ts_InPendantMode := FALSE;

// Clear reqs that may result in motion or physical changes to an axis
ClearMotionReqs;
// Clear other requests
ClearNonMotionReqs;

// Init fb with low reqs so rising edge detection is ready
procManualAxisReqsSpindle();
procManualAxisReqsOutE();
procManualAxisReqsInE();
procManualAxisReqsZ();
procManualAxisReqsHw();
procManualAxisReqsCfVfd();
END_ACTION
TRANSITION EMO Cmd FROM Stp_PendantMode TO Stp_EMOMode:=
// EStop command from safety plc H:Ok, L:EMO
NOT fs_EmoCmd
END_TRANSITION
(* @SFCISJUMP := 'Stp_EMOMode' *)
TRANSITION key not in run or bad SL FROM Stp_PendantMode TO Stp_SafeMode:=
// Keyswitch not in run or not okay, or not adequate security level
NOT fs_KeyswitchInRun OR
NOT fs_KeyswitchOk OR
operatingMode.SecurityLevel = SL_UNKNOWN OR
operatingMode.SecurityLevel = SL_GUEST
END_TRANSITION
TRANSITION req mode change FROM Stp_PendantMode TO Stp_CheckModeReq:=
// Keyswitch in run and adequate security level
fs_KeyswitchInRun AND
fs_KeyswitchOk AND
operatingMode.SecurityLevel >= SL_OPERATOR AND
// Req mode change (req other than current mode)
operatingMode.ModeReqBits <> 0 AND
(operatingMode.ModeReqBits AND OM_PENDANT_MODE) = 0

END_TRANSITION
(* @SFCISJUMP := 'Stp_CheckModeReq' *)
TRANSITION req production mode FROM Stp_CheckModeReq TO Stp_ProductionMode:=
// Keyswitch in run and adequate security level
fs_KeyswitchInRun AND
fs_KeyswitchOk AND
operatingMode.SecurityLevel >= SL_OPERATOR AND
// Req Production Mode
((operatingMode.ModeReqBits AND OM_PRODUCTION_MODE) <> 0) AND
// gate must be closed for production mode
fs_CfGateClosed
END_TRANSITION
STEP Stp_ProductionMode:
// Block mode request for current mode, but keep the others
// This prevents it from being seen as a request
operatingMode.ModeReqBits := operatingMode.ModeReqBits AND NOT OM_PRODUCTION_MODE; (* bit 6 clear *)

// Axis permit and other permissives
ProductionModeAxisPermits;
ModeIndependentPermissions;

// Decode HMI Submode
operatingMode.SubMode := fctDecodeHmiSubMode(operatingMode.HmiSubMode);

// Pulse the Reset SafeMC on request.
// This allows the reset of the safety enable instructions in the
// SafePLC while the system is not in EMO mode.
// The SafeMC reset sometimes isn't effective unless the axis is otherwise allowed to be powered.
tmrResetPulse(IN:= operatingMode.ReqEmoReset);
ts_ResetSafeMC := tmrResetPulse.Q;
operatingMode.ReqEmoReset := FALSE;

// In production mode, cycle start/stop on PB or HMI Req, or on cycle permissives not allowed to run
// Cycle Stop
// Stop PB held in or not okay keeps req stop high - blocking the start
tmrReqStopPulse(IN:= operatingMode.HmiReqCycleStop, PT:= T#500ms);
operatingMode.ReqCycleStop := (NOT fs_StopPbOk OR NOT fs_StopPbActive OR NOT cyclePermissives.allowCycleRun) OR tmrReqStopPulse.Q; // PB is L=stop
operatingMode.HmiReqCycleStop :=FALSE;

// Cycle Start
// Stop wins if start and stop are both active.
// Start on not stop and hmi or PB press and PB Okay.
// Start PB needs to be released to get a second pulse
tmrReqStartPulse(IN:= ((operatingMode.HmiReqCycleStart OR (fs_StartPbOk AND fs_StartPbActive)) AND cyclePermissives.allowCycleRun), PT:= T#20ms);
operatingMode.ReqCycleStart := NOT operatingMode.ReqCycleStop AND tmrReqStartPulse.Q;
operatingMode.HmiReqCycleStart :=FALSE;

// process the process requests
procHmiProcessReqs();
END_STEP
ENTRY_ACTION
// Set Operating State
operatingMode.OperatingMode := OM_PRODUCTION_MODE;
// To Safety PLC
ts_InProductionMode := TRUE;

// Clear process reqs on entry -- just in case one is spuriously set
ClearProcessReqs;

// Reset pulse timer
tmrResetPulse(IN:= FALSE, PT:= timeResetPulse);
END_ACTION
EXIT_ACTION
// To Safety PLC
ts_InProductionMode := FALSE;
END_ACTION
TRANSITION EMO Cmd FROM Stp_ProductionMode TO Stp_EMOMode:=
// EStop command from safety plc H:Ok, L:EMO
NOT fs_EmoCmd
END_TRANSITION
(* @SFCISJUMP := 'Stp_EMOMode' *)
TRANSITION key not in run or bad SL FROM Stp_ProductionMode TO Stp_SafeMode:=
// Keyswitch not in run or not okay, or not adequate security level
NOT fs_KeyswitchInRun OR
NOT fs_KeyswitchOk OR
operatingMode.SecurityLevel = SL_UNKNOWN OR
operatingMode.SecurityLevel = SL_GUEST
END_TRANSITION
TRANSITION req mode change FROM Stp_ProductionMode TO Stp_CheckModeReq:=
// Keyswitch in run and adequate security level
fs_KeyswitchInRun AND
fs_KeyswitchOk AND
operatingMode.SecurityLevel >= SL_OPERATOR AND
// Req mode change (req other than current mode)
operatingMode.ModeReqBits <> 0 AND
(operatingMode.ModeReqBits AND OM_PRODUCTION_MODE) = 0

END_TRANSITION
(* @SFCISJUMP := 'Stp_CheckModeReq' *)
STEP Stp_SafeMode:
// Clear mode requests if not ready to leave -- this guards against a lingering req
// being acted on long after it was issued, once conditions become okay to leave
IF NOT fs_KeyswitchInRun OR
    NOT fs_KeyswitchOk OR
    operatingMode.SecurityLevel < SL_OPERATOR THEN // OR
    // NOT fs_CfGateClosed THEN
  operatingMode.ModeReqBits := 16#0;
END_IF;

// Clear reqs that may result in motion or physical changes to an axis
ClearMotionReqs;
// Allow the other reqs (resets and set limits)

// Axis permit and other permissives
OtherModeAxisPermits;
ModeIndependentPermissions;

// Clear the other HMI Reqs
ClearCycleReqs;

END_STEP
ENTRY_ACTION
// Set Operating State
operatingMode.OperatingMode := OM_SAFE_MODE;
// To Safety PLC
ts_InSafeMode := TRUE;
// Initially clear the mode requests.
// They will be allowed once in the mode, and the keyswitch is in the run position
operatingMode.ModeReqBits := 16#0;

END_ACTION
EXIT_ACTION
// To Safety PLC
ts_InSafeMode := FALSE;
END_ACTION
TRANSITION EMO or Run and Mode Req FROM Stp_SafeMode TO Stp_CheckModeReq:=
// EStop command from safety plc H:Ok, L:EMO
NOT fs_EmoCmd OR
(
// Keyswitch in run and adequate security level
fs_KeyswitchInRun AND
fs_KeyswitchOk AND
operatingMode.SecurityLevel >= SL_OPERATOR AND
// Req Another Mode
// Leaving out of safe or emo will lock the gate,
// but the latched check is for production mode only.
((operatingMode.ModeReqBits AND OM_MANUAL_MODE) <> 0) OR
((operatingMode.ModeReqBits AND OM_PENDANT_MODE) <> 0) OR
((operatingMode.ModeReqBits AND OM_PRODUCTION_MODE) <> 0)
)

END_TRANSITION
(* @SFCISJUMP := 'Stp_CheckModeReq' *)
STEP Stp_EMOMode:

// clear mode requests while in EMO
operatingMode.ModeReqBits := 16#0;

// Axis permit and other permissives
OtherModeAxisPermits;
ModeIndependentPermissions;

// Clear reqs that may result in motion or physical changes to an axis
ClearMotionReqs;
// Clear other requests
ClearNonMotionReqs;

// Block cycle start/stop req in Emo
operatingMode.ReqCycleStart := FALSE;
operatingMode.ReqCycleStop := FALSE;
// Clear the reqs, but allow the EMO/Axis Reset ... they get handled below
operatingMode.HmiReqCycleStart := FALSE;
operatingMode.HmiReqCycleStop := FALSE;

// Run emo allow timer
// Only allow resets to emo if this timer is expired.
// If an e-stop removes power from the drives, it is bad for the drive power supplies to be
// energized less than 2 minutes after being deenergized -- capacitor discharge/recharge issue
tmrEStopResetAllow(IN:= TRUE);

// Clear the EMO reset bit if within this time
IF NOT tmrEStopResetAllow.Q THEN
  operatingMode.ReqEmoReset := FALSE;
END_IF;

// Calc how many seconds remain before a reset is allowed
eStopResetAllowSecRemain := TIME_TO_DINT(timeEStopResetAllow - tmrEStopResetAllow.ET) / 1000;

// We can't leave this state until EMO is clear, but we need the reset pulse to clear the EMO.
// If a reset request is received, send a reset pulse to the safe controller. In the event of
// multiple emo events, this may or may not clear all of them, but the status on the HMI should
// be updated, allowing the operators to see what else is needed.
// Run the reset pulse and send the reset req
tmrResetPulse(IN:= operatingMode.ReqEmoReset, PT:= timeResetPulse);
ts_ResetEStop := tmrResetPulse.Q;
operatingMode.ReqEmoReset := FALSE;

END_STEP
ENTRY_ACTION
// Set Operating State
operatingMode.OperatingMode := OM_EMO_MODE;

// To safety PLC
ts_InEmoMode := TRUE;

// Reset emo allow timer
tmrEStopResetAllow(IN:= FALSE, PT := timeEStopResetAllow);

END_ACTION
TRANSITION no emo, allow time done and reset req FROM Stp_EMOMode TO Stp_ResetAxes:=
// No more EMO, reset allow timer has expired, reset pulse is done
fs_EmoCmd AND
tmrEStopResetAllow.Q AND
// Use the reset pulse to the safe controller being done as time to leave instead of the request.
// This allows a request to create a pulse, and then be cleared.
// Meanwhile, the EMO may or may not clear, and the reset pulse will go away. If the EMO is gone
// when the reset pulse goes away, we can leave.
NOT ts_ResetEStop
END_TRANSITION
STEP Stp_ResetAxes:
// Clear mode requests while in EMO
operatingMode.ModeReqBits := 16#0;

// Run the reset pulse and send the reset req
tmrResetPulse(IN:= TRUE, PT:= timeResetPulse);
ts_ResetSafeMC := tmrResetPulse.Q;

END_STEP
ENTRY_ACTION
// Reset pulse timer
tmrResetPulse(IN:= FALSE, PT:= timeResetPulse);
END_ACTION
EXIT_ACTION
// To safety PLC
ts_InEmoMode := FALSE;

// Clear reqs that may result in motion or physical changes to an axis
ClearMotionReqs;
// Clear other requests
ClearNonMotionReqs;

// Clear other reqs
ClearCycleReqs;

END_ACTION
TRANSITION axis reset pulse done FROM Stp_ResetAxes TO Stp_SafeMode:=
// Emo Reset pulse complete
tmrResetPulse.ET = tmrResetPulse.PT AND NOT ts_ResetSafeMC
END_TRANSITION
(* @SFCISJUMP := 'Stp_SafeMode' *)
END_PROGRAM
```

#### Action.st
```iecst
ACTION ClearMotionReqs :
  // Clear Process Reqs, and then the machine specific axis Reqs
  // Process Reqs
  // Bool reqs
  pSrc := ADR(hmiProcessReqs.zReqMoveUpLimit);
  pDest := ADR(hmiProcessReqs.cuttingHeadMoveReqRetract);
  byteCount := pDest - pSrc + SIZEOF(BOOL);
  nxtAddr := brsmemset(pSrc, 0, byteCount);
  // Numerical reqs
  hmiProcessReqs.cuttingHeadReqDepth := 0.0;

  // Now clear the machine specific axis reqs
  FOR axisNo := 0 TO AXIS_COUNT DO
    // Bool reqs
    // (none)
    // numerical requests
    // (none)
    // move type and direction
    hmiMachineAxisReqs[axisNo].moveDesignation := -1; (* clear HMI selection *)
    hmiMachineAxisReqs[axisNo].direction := -1; (* clear HMI selection *)

    // Now clear the library requests
    // Bool reqs
    pSrc := ADR(hmiLibraryAxisReqs[axisNo].moveReq);
    pDest := ADR(hmiLibraryAxisReqs[axisNo].disengageSlaveReq);
    byteCount := pDest - pSrc + SIZEOF(BOOL);
    nxtAddr := brsmemset(pSrc, 0, byteCount);
    // numerical requests
    hmiLibraryAxisReqs[axisNo].Position := 0.0;
    hmiLibraryAxisReqs[axisNo].Distance := 0.0;
    hmiLibraryAxisReqs[axisNo].Velocity := 0.0;
    // move type and direction
    hmiLibraryAxisReqs[axisNo].moveDesignation := GAMOT_MD_NO_MOVE_COMMANDED;
    hmiLibraryAxisReqs[axisNo].Direction := mcDIR_UNDEFINED;
  END_FOR;

END_ACTION

ACTION ClearNonMotionReqs :
  // Clear the non-motion reqs
  FOR axisNo := 0 TO AXIS_COUNT DO
    // Clear requests to set limits and requests to reset
    // Bool reqs
    pSrc := ADR(hmiLibraryAxisReqs[axisNo].setPositionLimitsReq);
    pDest := ADR(hmiLibraryAxisReqs[axisNo].driveResetReq);
    byteCount := pDest - pSrc + SIZEOF(BOOL);
    nxtAddr := brsmemset(pSrc, 0, byteCount);
    // numerical requests
    // (none)
  END_FOR;

END_ACTION

ACTION ClearCycleReqs :
  // TODO: Does Cycle start/stop have a meaning in manual mode?
  // For now block them
  operatingMode.ReqCycleStart := FALSE;
  operatingMode.ReqCycleStop := FALSE;
  operatingMode.HmiReqCycleStart := FALSE;
  operatingMode.HmiReqCycleStop:= FALSE;
  operatingMode.ReqEmoReset := FALSE;
  operatingMode.ReqAxisReset := FALSE;
END_ACTION

ACTION ManualModeAxisPermits :
  // In Manual Mode
  // cycle is not okay to run
  cyclePermissives.isOmOk := FALSE;

  // TODO: Proper permissions. For now, wide open
  axes[AD_SPINDLE].MoveParameters.PosMovePermissive := TRUE;
  axes[AD_SPINDLE].MoveParameters.NegMovePermissive := TRUE;

  axes[AD_OUTER_ECCENTRIC].MoveParameters.PosMovePermissive := TRUE;
  axes[AD_OUTER_ECCENTRIC].MoveParameters.NegMovePermissive := TRUE;

  axes[AD_INNER_ECCENTRIC].MoveParameters.PosMovePermissive := TRUE;
  axes[AD_INNER_ECCENTRIC].MoveParameters.NegMovePermissive := TRUE;

  axes[AD_Z].MoveParameters.PosMovePermissive := TRUE;
  axes[AD_Z].MoveParameters.NegMovePermissive := TRUE;

  // Handwheel is virtual -- don't allow moves
  axes[AD_HANDWHEEL].MoveParameters.PosMovePermissive := FALSE;
  axes[AD_HANDWHEEL].MoveParameters.NegMovePermissive := FALSE;

  // cutting fluid pump
  axes[AD_CF_VFD].MoveParameters.PosMovePermissive := cfVfd.isAllowedToRun;
// Allow forward running only
  axes[AD_CF_VFD].MoveParameters.NegMovePermissive := FALSE;

END_ACTION

ACTION PendantModeAxisPermits :
    // In Pendant Mode
    // cycle is not okay to run
  cyclePermissives.isOmOk := FALSE;

  // TODO: Proper permissions. For now, wide open
  axes[AD_SPINDLE].MoveParameters.PosMovePermissive := TRUE;
  axes[AD_SPINDLE].MoveParameters.NegMovePermissive := TRUE;

  axes[AD_OUTER_ECCENTRIC].MoveParameters.PosMovePermissive := TRUE;
  axes[AD_OUTER_ECCENTRIC].MoveParameters.NegMovePermissive := TRUE;

  axes[AD_INNER_ECCENTRIC].MoveParameters.PosMovePermissive := TRUE;
  axes[AD_INNER_ECCENTRIC].MoveParameters.NegMovePermissive := TRUE;

  axes[AD_Z].MoveParameters.PosMovePermissive := TRUE;
  axes[AD_Z].MoveParameters.NegMovePermissive := TRUE;

  // Handwheel is virtual -- don't allow moves
  axes[AD_HANDWHEEL].MoveParameters.PosMovePermissive := FALSE;
  axes[AD_HANDWHEEL].MoveParameters.NegMovePermissive := FALSE;

  // cutting fluid pump
  axes[AD_CF_VFD].MoveParameters.PosMovePermissive := cfVfd.isAllowedToRun;
// Allow forward running only
  axes[AD_CF_VFD].MoveParameters.NegMovePermissive := FALSE;

END_ACTION

ACTION ProductionModeAxisPermits :
  // In Production Mode
  // cycle is okay to run
  cyclePermissives.isOmOk := TRUE;

  // Spindle
  // TODO: mask requests or commands?
  // fctClearMotionRequests(_I_ReqMask := MACM_NOMASK, _IO_Commands := axes[AD_SPINDLE].Commands);
  // Spindle is allowed to move forward as long as the cutting fluid is running
  // Spindle cannot run backward
  axes[AD_SPINDLE].MoveParameters.PosMovePermissive := cfVfd.isRunning AND cfVfd.isFlowEstablished;
  axes[AD_SPINDLE].MoveParameters.NegMovePermissive := FALSE;

  // Outer Eccentric
  // TODO: mask requests or commands?
  // fctClearMotionRequests(_I_ReqMask := MACM_NOMASK, _IO_Commands := axes[AD_OUTER_ECCENTRIC].Commands);
  // TODO: require spindle to be moving?
  axes[AD_OUTER_ECCENTRIC].MoveParameters.PosMovePermissive := TRUE;
  axes[AD_OUTER_ECCENTRIC].MoveParameters.NegMovePermissive := TRUE;
  // TODO: mask requests or commands?

  // Inner Eccentric
  // TODO: mask requests or commands?
  // fctClearMotionRequests(_I_ReqMask := MACM_NOMASK, _IO_Commands := axes[AD_INNER_ECCENTRIC].Commands);
  axes[AD_INNER_ECCENTRIC].MoveParameters.PosMovePermissive := TRUE;
  axes[AD_INNER_ECCENTRIC].MoveParameters.NegMovePermissive := TRUE;
  // TODO: mask requests or commands?

  // Z
  // TODO: mask requests or commands?
  // fctClearMotionRequests(_I_ReqMask := MACM_NOMASK, _IO_Commands := axes[AD_Z].Commands);
  // TODO: require eccentrics to be homed and spindle to be stopped
  axes[AD_Z].MoveParameters.PosMovePermissive := TRUE;
  axes[AD_Z].MoveParameters.NegMovePermissive := TRUE;
  // TODO: mask requests or commands?

  // Handwheel is virtual -- don't allow moves
  axes[AD_HANDWHEEL].MoveParameters.PosMovePermissive := FALSE;
  axes[AD_HANDWHEEL].MoveParameters.NegMovePermissive := FALSE;

  // cutting fluid pump
  axes[AD_CF_VFD].MoveParameters.PosMovePermissive := cfVfd.isAllowedToRun;
// Allow forward running only
  axes[AD_CF_VFD].MoveParameters.NegMovePermissive := FALSE;

END_ACTION

ACTION OtherModeAxisPermits:
    // Not in a mode (safe, initial, unknown, etc.)
    // This is some sort of error -- don't allow any motion
    // For each axis clear the requestes, and the move permissives
    // TODO: Clear the commnads?

    // cycle is no okay to run
  cyclePermissives.isOmOk := FALSE;

  // Spindle
  fctClearMotionRequests(_I_ReqMask := MACM_NOMASK, _IO_Commands := axes[AD_SPINDLE].Commands);
  // TODO: Clear the commnads, or let the axis SM handle it?
  // fctClearMotionCommands(_I_CmdMask := MACM_NOMASK, _IO_Commands := axes[AD_SPINDLE].Commands);
  axes[AD_SPINDLE].MoveParameters.PosMovePermissive := FALSE;
  axes[AD_SPINDLE].MoveParameters.NegMovePermissive := FALSE;

  // Outer Eccentric
  fctClearMotionRequests(_I_ReqMask := MACM_NOMASK, _IO_Commands := axes[AD_OUTER_ECCENTRIC].Commands);
  // TODO: Clear the commnads, or let the axis SM handle it?
  // fctClearMotionCommands(_I_CmdMask := MACM_NOMASK, _IO_Commands := axes[AD_OUTER_ECCENTRIC].Commands);
  axes[AD_OUTER_ECCENTRIC].MoveParameters.PosMovePermissive := FALSE;
  axes[AD_OUTER_ECCENTRIC].MoveParameters.NegMovePermissive := FALSE;

  // Inner Eccentric
  fctClearMotionRequests(_I_ReqMask := MACM_NOMASK, _IO_Commands := axes[AD_INNER_ECCENTRIC].Commands);
  // TODO: Clear the commnads, or let the axis SM handle it?
  // fctClearMotionCommands(_I_CmdMask := MACM_NOMASK, _IO_Commands := axes[AD_INNER_ECCENTRIC].Commands);
  axes[AD_INNER_ECCENTRIC].MoveParameters.PosMovePermissive := FALSE;
  axes[AD_INNER_ECCENTRIC].MoveParameters.NegMovePermissive := FALSE;

  // Z
  fctClearMotionRequests(_I_ReqMask := MACM_NOMASK, _IO_Commands := axes[AD_Z].Commands);
  // TODO: Clear the commnads, or let the axis SM handle it?
  // fctClearMotionCommands(_I_CmdMask := MACM_NOMASK, _IO_Commands := axes[AD_Z].Commands);
  axes[AD_Z].MoveParameters.PosMovePermissive := FALSE;
  axes[AD_Z].MoveParameters.NegMovePermissive := FALSE;

  // cutting fluid pump
  axes[AD_CF_VFD].MoveParameters.PosMovePermissive := cfVfd.isAllowedToRun;
// Allow forward running only
  axes[AD_CF_VFD].MoveParameters.NegMovePermissive := FALSE;

END_ACTION

ACTION ModeIndependentPermissions :
  // Set status and permissive related things that are independent of mode

  // Rollup of cycle start  allowed
  cyclePermissives.allowCycleStart :=
  // Operating mode must be okay
  cyclePermissives.isOmOk AND
  // Cutting fluid must be okay to start
  cfVfd.isAllowedToStart AND
    // Each axis needs to be in standstill or disabled. Additionally, inner eccentric can be coupled.
  (axes[AD_SPINDLE].Status.PlcOpenState = mcAXIS_DISABLED OR axes[AD_SPINDLE].Status.PlcOpenState = mcAXIS_STANDSTILL) AND
  (axes[AD_OUTER_ECCENTRIC].Status.PlcOpenState = mcAXIS_DISABLED OR axes[AD_OUTER_ECCENTRIC].Status.PlcOpenState = mcAXIS_STANDSTILL) AND
  (axes[AD_INNER_ECCENTRIC].Status.PlcOpenState = mcAXIS_DISABLED OR axes[AD_INNER_ECCENTRIC].Status.PlcOpenState = mcAXIS_STANDSTILL OR axes[AD_INNER_ECCENTRIC].Status.PlcOpenState = mcAXIS_SYNCHRONIZED_MOTION) AND
  (axes[AD_Z].Status.PlcOpenState = mcAXIS_DISABLED OR axes[AD_Z].Status.PlcOpenState = mcAXIS_STANDSTILL) AND
  // axes need to be referenced, and not force to be re-referenced
  axes[AD_SPINDLE].Status.IsHomed AND NOT axes[AD_SPINDLE].ForceSetRef AND
  axes[AD_OUTER_ECCENTRIC].Status.IsHomed AND NOT axes[AD_OUTER_ECCENTRIC].ForceSetRef AND
  axes[AD_INNER_ECCENTRIC].Status.IsHomed AND NOT axes[AD_INNER_ECCENTRIC].ForceSetRef AND
  axes[AD_Z].Status.IsHomed AND NOT axes[AD_Z].ForceSetRef AND
  // axes need to be calibrated to the process
  // Z will be indexed when the cycle is started, so no need to check it here, as long as Z is calibrated
  gr_PartCurrent.isZCalibrated AND gr_PartCurrent.isInECalibrated AND gr_PartCurrent.isOutECalibrated;

  // Rollup of cycle run allowed
  cyclePermissives.allowCycleRun :=
  // Operating mode must be okay
  cyclePermissives.isOmOk AND
  // Cutting fluid must be okay to start
  cfVfd.isAllowedToStart AND
    // Axes can't be in error or homing. Disabled is allowed because the cycle may start with them disabled.
  (axes[AD_SPINDLE].Status.PlcOpenState <> mcAXIS_ERRORSTOP AND axes[AD_SPINDLE].Status.PlcOpenState <> mcAXIS_HOMING) AND
  (axes[AD_OUTER_ECCENTRIC].Status.PlcOpenState <> mcAXIS_ERRORSTOP AND axes[AD_OUTER_ECCENTRIC].Status.PlcOpenState <> mcAXIS_HOMING) AND
  (axes[AD_INNER_ECCENTRIC].Status.PlcOpenState <> mcAXIS_ERRORSTOP AND axes[AD_INNER_ECCENTRIC].Status.PlcOpenState <> mcAXIS_HOMING) AND
  (axes[AD_Z].Status.PlcOpenState <> mcAXIS_ERRORSTOP AND axes[AD_Z].Status.PlcOpenState <> mcAXIS_HOMING) AND
  // axes need to be referenced, and not force to be re-referenced
  axes[AD_SPINDLE].Status.IsHomed AND NOT axes[AD_SPINDLE].ForceSetRef AND
  axes[AD_OUTER_ECCENTRIC].Status.IsHomed AND NOT axes[AD_OUTER_ECCENTRIC].ForceSetRef AND
  axes[AD_INNER_ECCENTRIC].Status.IsHomed AND NOT axes[AD_INNER_ECCENTRIC].ForceSetRef AND
  axes[AD_Z].Status.IsHomed AND NOT axes[AD_Z].ForceSetRef AND
  // axes need to be calibrated to the process
  // Z will be indexed when the cycle is started, so no need to check it here, as long as Z is calibrated
  gr_PartCurrent.isZCalibrated AND gr_PartCurrent.isInECalibrated AND gr_PartCurrent.isOutECalibrated;
END_ACTION
```

#### LocalFunctions.fun
```iecst
(* This function block will turn process requests into GaMpMotion library requests.
The GA Motion Library requests will then be handled by the fbHandleHmiAxisReq fb.
In this way, there is a cascading mechanism to get process specific then
machine specific then axis specific reqeusts processed by standard library functions,
even when process or machine specific things are not known by the library functions. *)
FUNCTION_BLOCK fbHandleHmiProcessReqs (* Turn process specific requests into GaMpMotion library requests. *)
  VAR_INPUT
    _I_ProcessReqs : REFERENCE TO sHmiProcessReqs;
    (* pointer to an array of sMot_HmiAxisReqs GA Motion Library requests *)
    (* use a pointer so array length does not need to known. *)
    _I_pLibraryAxesReqs : REFERENCE TO UDINT;
  END_VAR

  VAR
    (* automatic dereferencing of pLIbraryAxesReqs is not performed since it is being used as a pointer*)
    (* use this var below to hold a reference to an individual array element *)
    libReqs : REFERENCE TO sMot_HmiAxisReqs;
  END_VAR
END_FUNCTION_BLOCK

(* This function block will turn machine specific requests into GaMpMotion library requests.
Machine axis requests will be turned into library requests, and finally
library requests will be called using the library fb.
In this way, there is a cascading mechanism to get machine specific then axis
specific reqeusts processed by standard library functions,
even when process or machine specific things are not known by the library functions. *)
FUNCTION_BLOCK fbHandleHmiAxisReq (* Turn machine specific reqs into GaMpMotion library requs, and then call library fb fbProcessHmiAxisReq. *)
  VAR_INPUT
    _I_MachineAxisReqs : REFERENCE TO sHmiAxisReqs;
    _I_LibraryAxisReqs : REFERENCE TO sMot_HmiAxisReqs;
    _I_Axis : REFERENCE TO sMot_Axis;
    _I_SlaveAxis : REFERENCE TO sMot_Axis;
    _I_AxisPositionLimits : REFERENCE TO sMot_PositionLimits;
  END_VAR

  VAR
    procLibraryReq : fbProcessHmiAxisReq; (* library function block to handle standard reqs built into library *)
  END_VAR
END_FUNCTION_BLOCK

(* The HMI can easily set values like 0, 1, 2 from radio buttons, but it is harder to set specific move type values *)
(* This function is intended to take an HMI selection and return a move type usable by the GaMpMotion library *)
FUNCTION fctDecodeHmiMoveType : eGAMOT_MOVE_DESIGNATION (* Take in an HMI move type and return a corresponding enum move designation *)
  VAR_INPUT
    _I_AxisIsEndless : BOOL;
    _I_MoveReq : DINT;
    _I_MoveDirection : McDirectionEnum;
  END_VAR
END_FUNCTION

(* The HMI can easily set values like 0, 1, 2 from radio buttons, but it is harder to set specific move type values *)
(* This function is intended to take an HMI selection and return a direction usable by the McAxis library *)
FUNCTION fctDecodeHmiDirection : McDirectionEnum (* Take in an HMI move type and return a corresponding enum move designation *)
  VAR_INPUT
    _I_DirectionReq : DINT;
  END_VAR
END_FUNCTION
```

#### LocalFunctions.st
```iecst
(* This function block will turn process requests into GaMpMotion library requests.
The GA Motion Library requests will then be handled by the fbHandleHmiAxisReq fb.
In this way, there is a cascading mechanism to get process specific then
machine specific then axis specific reqeusts processed by standard library functions,
even when process or machine specific things are not known by the library functions. *)
FUNCTION_BLOCK fbHandleHmiProcessReqs (* Turn process specific requests into GaMpMotion library requests. *)
  // library axis req pointer is set ... assume it points to the first element of an array of sMot_HmiAxisReqs structures *)
  // TODO: Need to figure out syntax for accessing individual array elements and implement fb
  // libReqs ACCESS ADR(_I_pLibraryAxesReqs) + (AD_Z * SIZEOF(sMot_HmiAxisReqs)); // Set to access the Z Axis
  RETURN;
END_FUNCTION_BLOCK

(* This function block will turn machine specific requests into GaMpMotion library requests.
Machine axis requests will be turned into library requests, and finally
library requests will be called using the library fb.
In this way, there is a cascading mechanism to get machine specific then axis
specific reqeusts processed by standard library functions,
even when process or machine specific things are not known by the library functions. *)
FUNCTION_BLOCK fbHandleHmiAxisReq // Condition HMI process specific, then machine specific, and then process them with GaMpMotion library fbProcessHmiAxisReq.
  // Map (decode) HMI move type and then direction that the GAMpMotion library will see.
  // Note the direction and move parameters allowd are be influenced by the move type.
  // Do this before processing the move request so values can be checked or used before issuing a move.

  // Endless Axes, or continuous rotary axes (spindle and eccentrics) in this case,
  // in theory can use pos, neg, or shortest path (NOT supported yet).
  // For absolute moves, but non-continuous axes (Z) don't have a specfied direction for absolute moves -- the
  // direction is inherent to the requested position.
  // Also, an absolute move does not need distance, and a relative move does not need a position.
  // A velocity move does not need either.
  // Set the enable bits of the move direction as appropriate
  IF _I_MachineAxisReqs.moveDesignation = 0 THEN // absolute
    // An absolute move does not use distance, only position
    _I_MachineAxisReqs.moveDistanceEnable := FALSE;
    _I_MachineAxisReqs.movePositionEnable := TRUE;
    // now look at the axis and decied on what directions are allowed.
    IF _I_Axis.isAxisEndless THEN
      // Endless axis, absolute move: forward, backward, and shortest (if supported) are allowed
      _I_MachineAxisReqs.directionPosEnable := TRUE;
      _I_MachineAxisReqs.directionNegEnable := TRUE;
      _I_MachineAxisReqs.directionShortestEnable := FALSE; // could be true, but shortest is not supported yet
      // If the selected direction is shortest, then clear the selection
      IF _I_MachineAxisReqs.direction = 2 THEN
        _I_MachineAxisReqs.direction := -1;
      END_IF;
    ELSE
      // For non-endless axis, direction is inferred by move position, so the operator does not choose it
      // Disable choices and clear the selection
      _I_MachineAxisReqs.directionPosEnable := FALSE;
      _I_MachineAxisReqs.directionNegEnable := FALSE;
      _I_MachineAxisReqs.directionShortestEnable := FALSE;
      _I_MachineAxisReqs.direction := -1;
    END_IF;
  ELSIF _I_MachineAxisReqs.moveDesignation = 1 THEN // relative
    // A relative move does not use position, only distance
    _I_MachineAxisReqs.moveDistanceEnable := TRUE;
    _I_MachineAxisReqs.movePositionEnable := FALSE;
    // All axes, relative move: forward and backward are viable selections
    _I_MachineAxisReqs.directionPosEnable := TRUE;
    _I_MachineAxisReqs.directionNegEnable := TRUE;
    _I_MachineAxisReqs.directionShortestEnable := FALSE;
    // If the selected direction is shortest, then clear the selection
    IF _I_MachineAxisReqs.direction = 2 THEN
      _I_MachineAxisReqs.direction := -1;
    END_IF;
  ELSIF _I_MachineAxisReqs.moveDesignation = 2 THEN // velocity
    // A velocity move does not use position or distance
    _I_MachineAxisReqs.moveDistanceEnable := FALSE;
    _I_MachineAxisReqs.movePositionEnable := FALSE;
    // All axes, velocity move: forward and backward are viable selections
    _I_MachineAxisReqs.directionPosEnable := TRUE;
    _I_MachineAxisReqs.directionNegEnable := TRUE;
    _I_MachineAxisReqs.directionShortestEnable := FALSE;
    // If the selected direction is shortest, then clear the selection
    IF _I_MachineAxisReqs.direction = 2 THEN
      _I_MachineAxisReqs.direction := -1;
    END_IF;
  ELSE
    // Not caught move type (error case).
    // Allow move direction so move type can be determined in the move velocity case
    _I_MachineAxisReqs.moveDistanceEnable := FALSE;
    _I_MachineAxisReqs.movePositionEnable := FALSE;
    _I_MachineAxisReqs.directionPosEnable := FALSE;
    _I_MachineAxisReqs.directionNegEnable := FALSE;
    _I_MachineAxisReqs.directionShortestEnable := FALSE;
    _I_MachineAxisReqs.direction := -1;
  END_IF;

  // Coordinated shift commands cannot be enabled unless:
  // 1) The slave is coordinated and InSync
  // 2) The master is moving
  // 3) A phase shift or offset shift is not underway
  _I_MachineAxisReqs.shiftEnable := _I_Axis.Status.IsCoordInSync AND
    _I_Axis.Status.IsMoveActive AND
    NOT _I_Axis.CouplingParameters.OffsetShiftCmd AND
    NOT _I_Axis.CouplingParameters.PhaseShiftCmd;

  // Now the direction options should be qualified, set the direction that the GAMpMotion library will see
  _I_LibraryAxisReqs.Direction := fctDecodeHmiDirection(_I_DirectionReq := _I_MachineAxisReqs.direction);

  // Decode the HMI move designation into one the GAMpMotion library will see
  _I_LibraryAxisReqs.moveDesignation := fctDecodeHmiMoveType(
  _I_AxisIsEndless := _I_Axis.isAxisEndless,
  _I_MoveReq := _I_MachineAxisReqs.moveDesignation,
  _I_MoveDirection := _I_LibraryAxisReqs.Direction
  );

  // The move type and direction have now been pre-processed. Call the library function to process the requests.
  procLibraryReq(_I_HmiAxisReq := ADR(_I_LibraryAxisReqs), _I_Axis := ADR(_I_Axis), _I_SlaveAxis := ADR(_I_SlaveAxis), _I_AxisPositionLimits := ADR(_I_AxisPositionLimits));

END_FUNCTION_BLOCK

// The HMI can easily set values like 0, 1, 2 from radio buttons for example, but it is harder to set specific move type values
// This function is intended to take an HMI selection and return a move type usable by the GaMpMotion library.
// In the velocity move type case, if axis is endless, a velocity move is used. If the axis is
// not endless, jog limit instructions are used so limits can be considered.
FUNCTION fctDecodeHmiMoveType
  // Absolute move: HMI Value 0, GaMpMotion library 16#40
  // Relative move: HMI Value 1, GaMpMotion library 16#20
  // Velocity move: HMI Value 2
  // Velocity GaMpMotion library 16#10
  // Jog Limit Up Fwd GaMpMotion library 16#04
  // Jog Limit Down Rev GaMpMotion library 16#08
  IF _I_MoveReq = 0 THEN
    fctDecodeHmiMoveType := GAMOT_MD_ABSOLUTE;
  ELSIF _I_MoveReq = 1 THEN
    fctDecodeHmiMoveType := GAMOT_MD_RELATIVE;
  ELSIF _I_MoveReq = 2 THEN
    // If the axis is endless, use a velocity move, otherwise use a Jog Limit move
    // The jog limit requires a direction so the correct instruction and limit can be considered.
    IF _I_AxisIsEndless THEN
      fctDecodeHmiMoveType := GAMOT_MD_VELOCITY;
    ELSE
      IF _I_MoveDirection = mcDIR_POSITIVE THEN
        fctDecodeHmiMoveType := GAMOT_MD_JOG_LIMIT_UP_FWD;
      ELSIF _I_MoveDirection = mcDIR_NEGATIVE THEN
        fctDecodeHmiMoveType := GAMOT_MD_JOG_LIMIT_DOWN_REV;
      ELSE
        fctDecodeHmiMoveType := GAMOT_MD_NO_MOVE_COMMANDED;
      END_IF;
    END_IF;
  ELSE
      fctDecodeHmiMoveType := GAMOT_MD_NO_MOVE_COMMANDED;
  END_IF;
END_FUNCTION

// The HMI can easily set values like 0, 1, 2 from radio buttons, but it is harder to set specific move type values
// This function is intended to take an HMI selection and return a direction usable by the McAxis library
FUNCTION fctDecodeHmiDirection
  // Positive Direction: HMI Value 0, GaMpMotion library 0
  // Negative Direction: HMI Value 1, GaMpMotion library 1
  // Shortest Path:      HMI Value 2, GaMpMotion library 3
  IF _I_DirectionReq = 0 THEN
    fctDecodeHmiDirection := mcDIR_POSITIVE;
  ELSIF _I_DirectionReq = 1 THEN
    fctDecodeHmiDirection := mcDIR_NEGATIVE;
  ELSIF _I_DirectionReq = 2 THEN
    fctDecodeHmiDirection := mcDIR_SHORTEST_WAY;
  ELSE
    fctDecodeHmiDirection := mcDIR_UNDEFINED;
  END_IF;
END_FUNCTION
```

#### OmSM - Copy.sfc - not listed in the package file held
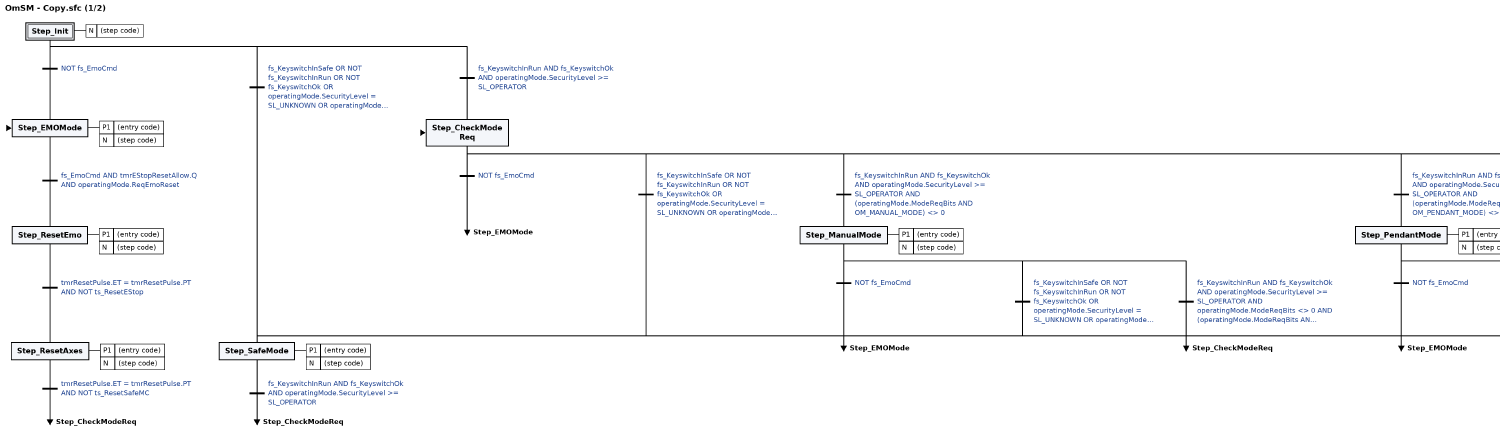
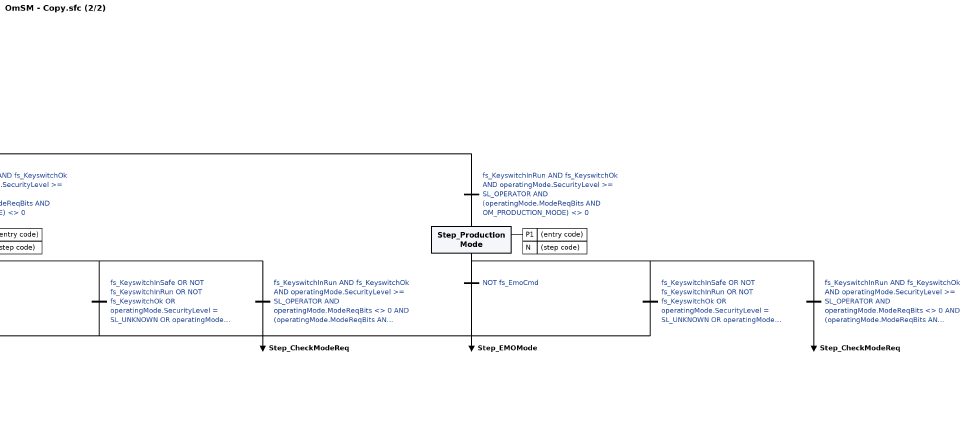
```iecst
PROGRAM _CYCLIC
INITIAL_STEP Step_Init:
// Set Operating State
operatingMode.OperatingMode := OM_INITIAL;
END_STEP
TRANSITION EMO Cmd FROM Step_Init TO Step_EMOMode:=
// EStop command from safety plc H:Ok, L:EMO
NOT fs_EmoCmd
END_TRANSITION
TRANSITION keyswich in safe, not ok or bad SL FROM Step_Init TO Step_SafeMode:=
// Keyswitch in safe, or not in run or not okay, or not adequate security level
fs_KeyswitchInSafe OR
NOT fs_KeyswitchInRun OR
NOT fs_KeyswitchOk OR
operatingMode.SecurityLevel = SL_UNKNOWN OR
operatingMode.SecurityLevel = SL_GUEST
END_TRANSITION
TRANSITION keyswitch in run and SL FROM Step_Init TO Step_CheckModeReq:=
// Keyswitch in run and adequate security level
fs_KeyswitchInRun AND
fs_KeyswitchOk AND
operatingMode.SecurityLevel >= SL_OPERATOR

END_TRANSITION
STEP Step_CheckModeReq:
END_STEP
TRANSITION EMO Cmd FROM Step_CheckModeReq TO Step_EMOMode:=
// EStop command from safety plc H:Ok, L:EMO
NOT fs_EmoCmd
END_TRANSITION
(* @SFCISJUMP := 'Step_EMOMode' *)
TRANSITION key not in run or bad SL FROM Step_CheckModeReq TO Step_SafeMode:=
// Keyswitch in safe, or not in run or not okay, or not adequate security level
fs_KeyswitchInSafe OR
NOT fs_KeyswitchInRun OR
NOT fs_KeyswitchOk OR
operatingMode.SecurityLevel = SL_UNKNOWN OR
operatingMode.SecurityLevel = SL_GUEST
END_TRANSITION
TRANSITION req manual mode FROM Step_CheckModeReq TO Step_ManualMode:=
// Keyswitch in run and adequate security level
fs_KeyswitchInRun AND
fs_KeyswitchOk AND
operatingMode.SecurityLevel >= SL_OPERATOR AND
// Req Manual Mode
(operatingMode.ModeReqBits AND OM_MANUAL_MODE) <> 0

END_TRANSITION
STEP Step_ManualMode:
// Block mode request for current mode
// This prevents it from being seen as a request
operatingMode.ModeReqBits := operatingMode.ModeReqBits XOR OM_MANUAL_MODE; (* bit 4 clear *)

END_STEP
ENTRY_ACTION
// Set Operating State
operatingMode.OperatingMode := OM_MANUAL_MODE;
END_ACTION
TRANSITION EMO Cmd FROM Step_ManualMode TO Step_EMOMode:=
// EStop command from safety plc H:Ok, L:EMO
NOT fs_EmoCmd
END_TRANSITION
(* @SFCISJUMP := 'Step_EMOMode' *)
TRANSITION key not in run or bad SL FROM Step_ManualMode TO Step_SafeMode:=
// Keyswitch in safe, or not in run or not okay, or not adequate security level
fs_KeyswitchInSafe OR
NOT fs_KeyswitchInRun OR
NOT fs_KeyswitchOk OR
operatingMode.SecurityLevel = SL_UNKNOWN OR
operatingMode.SecurityLevel = SL_GUEST
END_TRANSITION
TRANSITION req mode change FROM Step_ManualMode TO Step_CheckModeReq:=
// Keyswitch in run and adequate security level
fs_KeyswitchInRun AND
fs_KeyswitchOk AND
operatingMode.SecurityLevel >= SL_OPERATOR AND
// Req mode change (req other than current mode)
operatingMode.ModeReqBits <> 0 AND
(operatingMode.ModeReqBits AND OM_MANUAL_MODE) = 0

END_TRANSITION
(* @SFCISJUMP := 'Step_CheckModeReq' *)
TRANSITION req pendnat mode FROM Step_CheckModeReq TO Step_PendantMode:=
// Keyswitch in run and adequate security level
fs_KeyswitchInRun AND
fs_KeyswitchOk AND
operatingMode.SecurityLevel >= SL_OPERATOR AND
// Req Pendant Mode
(operatingMode.ModeReqBits AND OM_PENDANT_MODE) <> 0
END_TRANSITION
STEP Step_PendantMode:
// Block mode request for current mode
// This prevents it from being seen as a request
operatingMode.ModeReqBits := operatingMode.ModeReqBits XOR OM_PENDANT_MODE; (* bit 5 clear *)
END_STEP
ENTRY_ACTION
// Set Operating State
operatingMode.OperatingMode := OM_PENDANT_MODE;
END_ACTION
TRANSITION EMO Cmd FROM Step_PendantMode TO Step_EMOMode:=
// EStop command from safety plc H:Ok, L:EMO
NOT fs_EmoCmd
END_TRANSITION
(* @SFCISJUMP := 'Step_EMOMode' *)
TRANSITION key not in run or bad SL FROM Step_PendantMode TO Step_SafeMode:=
// Keyswitch in safe, or not in run or not okay, or not adequate security level
fs_KeyswitchInSafe OR
NOT fs_KeyswitchInRun OR
NOT fs_KeyswitchOk OR
operatingMode.SecurityLevel = SL_UNKNOWN OR
operatingMode.SecurityLevel = SL_GUEST
END_TRANSITION
TRANSITION req mode change FROM Step_PendantMode TO Step_CheckModeReq:=
// Keyswitch in run and adequate security level
fs_KeyswitchInRun AND
fs_KeyswitchOk AND
operatingMode.SecurityLevel >= SL_OPERATOR AND
// Req mode change (req other than current mode)
operatingMode.ModeReqBits <> 0 AND
(operatingMode.ModeReqBits AND OM_PENDANT_MODE) = 0
END_TRANSITION
(* @SFCISJUMP := 'Step_CheckModeReq' *)
TRANSITION req production mode FROM Step_CheckModeReq TO Step_ProductionMode:=
// Keyswitch in run and adequate security level
fs_KeyswitchInRun AND
fs_KeyswitchOk AND
operatingMode.SecurityLevel >= SL_OPERATOR AND
// Req Production Mode
(operatingMode.ModeReqBits AND OM_PRODUCTION_MODE) <> 0
END_TRANSITION
STEP Step_ProductionMode:
// Block mode request for current mode
// This prevents it from being seen as a request
operatingMode.ModeReqBits := operatingMode.ModeReqBits XOR OM_PRODUCTION_MODE; (* bit 6 clear *)
END_STEP
ENTRY_ACTION
// Set Operating State
operatingMode.OperatingMode := OM_PRODUCTION_MODE;
END_ACTION
TRANSITION EMO Cmd FROM Step_ProductionMode TO Step_EMOMode:=
// EStop command from safety plc H:Ok, L:EMO
NOT fs_EmoCmd
END_TRANSITION
(* @SFCISJUMP := 'Step_EMOMode' *)
TRANSITION key not in run or bad SL FROM Step_ProductionMode TO Step_SafeMode:=
// Keyswitch in safe, or not in run or not okay, or not adequate security level
fs_KeyswitchInSafe OR
NOT fs_KeyswitchInRun OR
NOT fs_KeyswitchOk OR
operatingMode.SecurityLevel = SL_UNKNOWN OR
operatingMode.SecurityLevel = SL_GUEST
END_TRANSITION
TRANSITION req mode change FROM Step_ProductionMode TO Step_CheckModeReq:=
// Keyswitch in run and adequate security level
fs_KeyswitchInRun AND
fs_KeyswitchOk AND
operatingMode.SecurityLevel >= SL_OPERATOR AND
// Req mode change (req other than current mode)
operatingMode.ModeReqBits <> 0 AND
(operatingMode.ModeReqBits AND OM_PRODUCTION_MODE) = 0

END_TRANSITION
(* @SFCISJUMP := 'Step_CheckModeReq' *)
STEP Step_SafeMode:
// clear mode requests while in safe
operatingMode.ModeReqBits := 16#0;
END_STEP
ENTRY_ACTION
// Set Operating State
operatingMode.OperatingMode := OM_SAFE_MODE;
END_ACTION
TRANSITION keyswitch in run and SL FROM Step_SafeMode TO Step_CheckModeReq:=
// Keyswitch in run and adequate security level
fs_KeyswitchInRun AND
fs_KeyswitchOk AND
operatingMode.SecurityLevel >= SL_OPERATOR

END_TRANSITION
(* @SFCISJUMP := 'Step_CheckModeReq' *)
STEP Step_EMOMode:
// clear mode requests while in EMO
operatingMode.ModeReqBits := 16#0;

// Run emo allow timer
// Only allow resets to emo if this timer is expired.
// If an e-stop removes power from the drives, it is bad for the drive power supplies to be
// energized less than 2 minutes after being deenergized -- capacitor discharge/recharge issue
tmrEStopResetAllow(IN:= TRUE, PT := timeEStopResetAllow);

// Clear the reset bits if within this time
IF NOT tmrEStopResetAllow.Q THEN
  operatingMode.ReqEmoReset := FALSE;
  operatingMode.ReqAxisReset := FALSE;
END_IF;

// Calc how many seconds remain before a reset is allowed
eStopResetAllowSecRemain := TIME_TO_DINT(timeEStopResetAllow - tmrEStopResetAllow.ET) / 1000;

END_STEP
ENTRY_ACTION
// Set Operating State
operatingMode.OperatingMode := OM_EMO_MODE;

// Reset emo allow timer
tmrEStopResetAllow(IN:= FALSE, PT := timeEStopResetAllow);

END_ACTION
TRANSITION no emo, allow time done and reset req FROM Step_EMOMode TO Step_ResetEmo:=
// No more EMO, reset allow timer has expired, and a reset is requested
fs_EmoCmd AND
tmrEStopResetAllow.Q AND
operatingMode.ReqEmoReset
END_TRANSITION
STEP Step_ResetEmo:
// Clear mode requests while in EMO
operatingMode.ModeReqBits := 16#0;

// Run the reset pulse and send the reset req
tmrResetPulse(IN:= TRUE, PT:= timeResetPulse);
ts_ResetEStop := tmrResetPulse.Q;
END_STEP
ENTRY_ACTION
// Reset pulse timer
tmrResetPulse(IN:= FALSE, PT:= timeResetPulse);
END_ACTION
TRANSITION emo reset pulse done FROM Step_ResetEmo TO Step_ResetAxes:=
// Emo Reset pulse complete
tmrResetPulse.ET = tmrResetPulse.PT AND NOT ts_ResetEStop
END_TRANSITION
STEP Step_ResetAxes:
// Clear mode requests while in EMO
operatingMode.ModeReqBits := 16#0;

// Run the reset pulse and send the reset req
tmrResetPulse(IN:= TRUE, PT:= timeResetPulse);
ts_ResetSafeMC := tmrResetPulse.Q;
END_STEP
ENTRY_ACTION
// Reset pulse timer
tmrResetPulse(IN:= FALSE, PT:= timeResetPulse);
END_ACTION
TRANSITION axis reset pulse done FROM Step_ResetAxes TO Step_CheckModeReq:=
// Emo Reset pulse complete
tmrResetPulse.ET = tmrResetPulse.PT AND NOT ts_ResetSafeMC
END_TRANSITION
(* @SFCISJUMP := 'Step_CheckModeReq' *)
END_PROGRAM
```

### Program Logical/PlcLogic/Annunc (IEC)

#### Annunc.var
```iecst
VAR CONSTANT

END_VAR

VAR
  tmr025Hz : TON; (* 0.25 Hz timer *)
  tmr050Hz : TON; (* 0.50 Hz timer *)
  tmr100Hz : TON; (* 1 Hz timer *)
END_VAR
```

#### Main.st
```iecst
PROGRAM _INIT
  tmr025Hz.PT := T#250ms;
  tmr050Hz.PT := T#500ms;
  tmr100Hz.PT := T#1000ms;
END_PROGRAM

PROGRAM _CYCLIC

  // Create blinking bits (global variables), 50% duty cycle
  // 0.25 Hz (4x/sec)
  tmr025Hz(IN:= NOT tmr025Hz.Q);
  IF tmr025Hz.Q THEN
    blink025Hz := NOT blink025Hz;
  END_IF;
  // 0.5 Hz (2x/sec)
  tmr050Hz(IN:= NOT tmr050Hz.Q);
  IF tmr050Hz.Q THEN
    blink050Hz := NOT blink050Hz;
  END_IF;
  // 1.0 Hz (1x/sec)
  tmr100Hz(IN:= NOT tmr100Hz.Q);
  IF tmr100Hz.Q THEN
    blink100Hz := NOT blink100Hz;
  END_IF;

  // Light the 480 VAC Okay lamp on the OWS if the power monitor in the MCP is okay.
  DO_PL_OWSAmber :=  DI_JI_480VACOk.Value;

END_PROGRAM

PROGRAM _EXIT
	(* Insert code here *)

END_PROGRAM
```

### Program Logical/PlcLogic/AxEnable (IEC)

#### AxEnable.st - Init, cyclic, exit code
```iecst
PROGRAM _INIT

END_PROGRAM

PROGRAM _CYCLIC

  // TODO: Decide when drives shall be enabled by the PLC
  // For now, enable them for easy initial testing.
  // H: Enable, L: Stop
  axes[AD_SPINDLE].Commands.PlcSafetyEnable := TRUE;
  axes[AD_OUTER_ECCENTRIC].Commands.PlcSafetyEnable := TRUE;
  axes[AD_INNER_ECCENTRIC].Commands.PlcSafetyEnable := TRUE;
  axes[AD_Z].Commands.PlcSafetyEnable := TRUE;

END_PROGRAM

PROGRAM _EXIT
	(* Insert code here *)

END_PROGRAM
```

### Program Logical/PlcLogic/ProdCycle (IEC)

#### ProdCycle.typ - Local data types
```iecst
TYPE
  ePROD_CYCLE_STEP :
    (
    PCS_UNKNOWN         := 0,
    PCS_INIT            := 1,
    PCS_MODE_CHECK      := 2,
    PCS_WAIT_FOR_PROD   := 3,
    PCS_WAIT_FOR_START  := 4,
    PCS_DECOUPLE_ECC    := 5,
    PCS_RESET_AXES      := 6,
    PCS_ENABLE_AXES     := 7,
    PCS_START_CF        := 8,
    PCS_ZERO_DEPTH      := 9,
    PCS_Z_TO_SOC        := 10,
    PCS_NEXT_CYCLE      := 11,
    PCS_START_SPINDLE   := 12,
    PCS_COUPLE_ECC      := 13,
    PCS_START_PASS      := 14,
    PCS_SYNCHING1       := 15,
    PCS_SYNCHING2       := 16,
    PCS_SYNCHING3       := 17,
    PCS_AXES_SYNCHED    := 18,
    PCS_SET_NEXT_PASS   := 19,
    PCS_SET_FINISH_PASS := 20,
    PCS_SET_RETRACT     := 21,
    PCS_STOP_SPINDLE    := 22,
    PCS_INDEX_Z_WAIT    := 23,
    PCS_CF_OFF1         := 24,
    PCS_CF_OFF2         := 25,
    PCS_Z_TO_UNLOAD     := 26,
    PCS_DONE_WAIT       := 27,
    PCS_INDEX_Z         := 28,
    PCS_EOC_WAIT        := 29,
    PCS_CF_TO           := 30,
    PCS_START_CF2       := 31,
    (* cycle stop related *)
    PCS_CYCLE_STOP      := 32,
    PCS_CS_STOP_AXES    := 33,
    PCS_CS_ZERO_DEPTH   := 34,
    PCS_CS_STOP_SPINDLE := 35,
    PCS_CS_DISABLE_AXES := 36,
    PCS_CS_STOP_CF      := 37
  ) := PCS_INIT;

 END_TYPE
```

#### ProdCycle.var - Local variables
```iecst
VAR CONSTANT

END_VAR

VAR RETAIN

END_VAR

VAR
  disableStepTO : BOOL := FALSE;
  startCycleOS : BOOL := FALSE;
  idx : SINT;

  tmrStepMin : TON; (* hold step for min time *)
  tmrStepTO : TON; (* step timeout timer *)
  tmrCfShutoff : TON; (* shutoff cooling pump after a delay *)
  fbCalcMoveTimes : fbCalcTrapMoveTime; (* function block to calculate trapazoidal move times *)

  (* info to safety controller *)
  ts_InCycle : BOOL; (* tell the safe controller we are in cycle *)
  ts_cfLockGate : BOOL; (* lock the cutting fluid gate *)

  (* production cycle step information *)
  (* indexes correspond to ePROD_CYCLE_STEP values *)
  (* move to global variables so they can be permanent *)
  (* stepETs  : ARRAY[0..40] OF TIME; step elapsed times *)
  (* stepIsTO : ARRAY[0..40] OF BOOL; set if the step has a TO *)

  prodCycleStep : ePROD_CYCLE_STEP;
END_VAR
```

#### Init.st
```iecst
PROGRAM _INIT
  // Init step TOs
  SetStepTOs; // not normally needed -- can rely on permanent variable nature

END_PROGRAM
```
